LIN {X 0,Y 580.3,Z 452.202,A -85,B 0,C 180,E1 -1946.144,E2 -1946.144} C_VEL
LIN {X 0,Y 580.268,Z 452.203,A -85,B 0,C 180,E1 -1948.614,E2 -1948.614} C_VEL
LIN {X 0,Y 580.272,Z 452.198,A -85,B 0,C 180,E1 -1951.022,E2 -1951.022} C_VEL
LIN {X 0,Y 580.272,Z 452.198,A -85,B 0,C 180,E1 -1953.666,E2 -1953.666} C_VEL
LIN {X 0,Y 580.251,Z 452.21,A -85,B 0,C 180,E1 -1956.441,E2 -1956.441} C_VEL
LIN {X 0,Y 580.254,Z 452.2,A -85,B 0,C 180,E1 -1959.436,E2 -1959.436} C_VEL
LIN {X 0,Y 580.242,Z 452.202,A -85,B 0,C 180,E1 -1961.644,E2 -1961.644} C_VEL
LIN {X 0,Y 580.251,Z 452.202,A -85,B 0,C 180,E1 -1963.825,E2 -1963.825} C_VEL
LIN {X 0,Y 580.255,Z 452.206,A -85,B 0,C 180,E1 -1966.695,E2 -1966.695} C_VEL
LIN {X 0,Y 580.293,Z 452.195,A -85,B 0,C 180,E1 -1969.533,E2 -1969.533} C_VEL
LIN {X 0,Y 580.321,Z 452.199,A -85,B 0,C 180,E1 -1972.344,E2 -1972.344} C_VEL
LIN {X 0,Y 580.315,Z 452.194,A -85,B 0,C 180,E1 -1975.137,E2 -1975.137} C_VEL
LIN {X 0,Y 580.312,Z 452.194,A -85,B 0,C 180,E1 -1977.918,E2 -1977.918} C_VEL
LIN {X 0,Y 580.36,Z 452.195,A -85,B 0,C 180,E1 -1980.694,E2 -1980.694} C_VEL
LIN {X 0,Y 580.267,Z 452.198,A -85,B 0,C 180,E1 -1983.472,E2 -1983.472} C_VEL
LIN {X 0,Y 580.306,Z 452.193,A -85,B 0,C 180,E1 -1985.56,E2 -1985.56} C_VEL
LIN {X 0,Y 580.319,Z 452.198,A -85,B 0,C 180,E1 -1988.356,E2 -1988.356} C_VEL
LIN {X 0,Y 580.319,Z 452.193,A -85,B 0,C 180,E1 -1991.208,E2 -1991.208} C_VEL
LIN {X 0,Y 580.3,Z 452.199,A -85,B 0,C 180,E1 -1994.339,E2 -1994.339} C_VEL
LIN {X 0,Y 580.298,Z 452.201,A -85,B 0,C 180,E1 -1996.914,E2 -1996.914} C_VEL
LIN {X 0,Y 580.293,Z 452.195,A -85,B 0,C 180,E1 -1999.822,E2 -1999.822} C_VEL
LIN {X 0,Y 580.272,Z 452.199,A -85,B 0,C 180,E1 -2001.35,E2 -2001.35} C_VEL
LIN {X 0,Y 579.575,Z 452.286,A -85,B 0,C 180,E1 -2001.929,E2 -2001.929} C_VEL
LIN {X 0,Y 576.696,Z 452.651,A -85,B 0,C 180,E1 -2002.869,E2 -2002.869} C_VEL
LIN {X 0,Y 574.301,Z 452.945,A -85,B 0,C 180,E1 -2003.625,E2 -2003.625} C_VEL
LIN {X 0,Y 573.303,Z 453.068,A -85,B 0,C 180,E1 -2004.209,E2 -2004.209} C_VEL
LIN {X 0,Y 573.237,Z 453.079,A -85,B 0,C 180,E1 -2004.406,E2 -2004.406} C_VEL
LIN {X 0,Y 573.242,Z 453.08,A -85,B 0,C 180,E1 -2006.976,E2 -2006.976} C_VEL
LIN {X 0,Y 573.236,Z 453.075,A -85,B 0,C 180,E1 -2009.489,E2 -2009.489} C_VEL
LIN {X 0,Y 573.243,Z 453.075,A -85,B 0,C 180,E1 -2012.23,E2 -2012.23} C_VEL
LIN {X 0,Y 573.241,Z 453.084,A -85,B 0,C 180,E1 -2014.775,E2 -2014.775} C_VEL
LIN {X 0,Y 573.241,Z 453.078,A -85,B 0,C 180,E1 -2017.167,E2 -2017.167} C_VEL
LIN {X 0,Y 573.236,Z 453.074,A -85,B 0,C 180,E1 -2019.608,E2 -2019.608} C_VEL
LIN {X 0,Y 573.232,Z 453.081,A -85,B 0,C 180,E1 -2022.643,E2 -2022.643} C_VEL
LIN {X 0,Y 573.228,Z 453.075,A -85,B 0,C 180,E1 -2025.668,E2 -2025.668} C_VEL
LIN {X 0,Y 573.251,Z 453.077,A -85,B 0,C 180,E1 -2028.547,E2 -2028.547} C_VEL
LIN {X 0,Y 573.241,Z 453.078,A -85,B 0,C 180,E1 -2031.3,E2 -2031.3} C_VEL
LIN {X 0,Y 573.234,Z 453.074,A -85,B 0,C 180,E1 -2034.015,E2 -2034.015} C_VEL
LIN {X 0,Y 573.276,Z 453.072,A -85,B 0,C 180,E1 -2036.52,E2 -2036.52} C_VEL
LIN {X 0,Y 573.233,Z 453.083,A -85,B 0,C 180,E1 -2039.117,E2 -2039.117} C_VEL
LIN {X 0,Y 573.258,Z 453.071,A -85,B 0,C 180,E1 -2041.969,E2 -2041.969} C_VEL
LIN {X 0,Y 573.248,Z 453.076,A -85,B 0,C 180,E1 -2044.591,E2 -2044.591} C_VEL
LIN {X 0,Y 573.232,Z 453.076,A -85,B 0,C 180,E1 -2047.663,E2 -2047.663} C_VEL
LIN {X 0,Y 573.273,Z 453.074,A -85,B 0,C 180,E1 -2050.729,E2 -2050.729} C_VEL
LIN {X 0,Y 573.255,Z 453.074,A -85,B 0,C 180,E1 -2053.623,E2 -2053.623} C_VEL
LIN {X 0,Y 573.27,Z 453.071,A -85,B 0,C 180,E1 -2055.808,E2 -2055.808} C_VEL
LIN {X 0,Y 573.26,Z 453.075,A -85,B 0,C 180,E1 -2058.746,E2 -2058.746} C_VEL
LIN {X 0,Y 573.288,Z 453.073,A -85,B 0,C 180,E1 -2061.542,E2 -2061.542} C_VEL
LIN {X 0,Y 573.295,Z 453.068,A -85,B 0,C 180,E1 -2064.373,E2 -2064.373} C_VEL
LIN {X 0,Y 573.313,Z 453.068,A -85,B 0,C 180,E1 -2067.894,E2 -2067.894} C_VEL
LIN {X 0,Y 573.342,Z 453.273,A -85,B 0,C 180,E1 -2070.462,E2 -2070.462} C_VEL
LIN {X 0,Y 573.575,Z 454.38,A -85,B 0,C 180,E1 -2070.572,E2 -2070.572} C_VEL
LIN {X 0,Y 574.043,Z 456.439,A -85,B 0,C 180,E1 -2070.615,E2 -2070.615} C_VEL
LIN {X 0,Y 573.909,Z 533.892,A -85,B 0,C 180,E1 -2071.602,E2 -2071.602} C_VEL
LIN {X 0,Y 573.777,Z 547.056,A -85,B 0,C 180,E1 -2071.91,E2 -2071.91} C_VEL
LIN {X 0,Y 573.683,Z 559.086,A -85,B 0,C 180,E1 -2072.327,E2 -2072.327} C_VEL
LIN {X 0,Y 573.567,Z 571.273,A -85,B 0,C 180,E1 -2072.898,E2 -2072.898} C_VEL
LIN {X 0,Y 573.429,Z 582.799,A -85,B 0,C 180,E1 -2073.602,E2 -2073.602} C_VEL
LIN {X 0,Y 573.315,Z 593.186,A -85,B 0,C 180,E1 -2074.395,E2 -2074.395} C_VEL
LIN {X 0,Y 573.24,Z 602.582,A -85,B 0,C 180,E1 -2075.277,E2 -2075.277} C_VEL
LIN {X 0,Y 573.148,Z 611.669,A -85,B 0,C 180,E1 -2076.337,E2 -2076.337} C_VEL
LIN {X 0,Y 573.107,Z 619.017,A -85,B 0,C 180,E1 -2077.399,E2 -2077.399} C_VEL
LIN {X 0,Y 573.056,Z 624.934,A -85,B 0,C 180,E1 -2078.464,E2 -2078.464} C_VEL
LIN {X 0,Y 572.993,Z 629.615,A -85,B 0,C 180,E1 -2079.532,E2 -2079.532} C_VEL
LIN {X 0,Y 573.009,Z 633.181,A -85,B 0,C 180,E1 -2080.603,E2 -2080.603} C_VEL
LIN {X 0,Y 572.975,Z 634.995,A -85,B 0,C 180,E1 -2081.319,E2 -2081.319} C_VEL
LIN {X 0,Y 572.946,Z 636.36,A -85,B 0,C 180,E1 -2082.037,E2 -2082.037} C_VEL
LIN {X 0,Y 572.945,Z 637.318,A -85,B 0,C 180,E1 -2082.757,E2 -2082.757} C_VEL
LIN {X 0,Y 572.968,Z 637.871,A -85,B 0,C 180,E1 -2083.478,E2 -2083.478} C_VEL
LIN {X 0,Y 572.942,Z 637.951,A -85,B 0,C 180,E1 -2084.292,E2 -2084.292} C_VEL
LIN {X 0,Y 572.916,Z 636.947,A -85,B 0,C 180,E1 -2085.658,E2 -2085.658} C_VEL
LIN {X 0,Y 572.943,Z 634.69,A -85,B 0,C 180,E1 -2086.906,E2 -2086.906} C_VEL
LIN {X 0,Y 572.997,Z 630.813,A -85,B 0,C 180,E1 -2088.227,E2 -2088.227} C_VEL
LIN {X 0,Y 573.042,Z 626.292,A -85,B 0,C 180,E1 -2089.339,E2 -2089.339} C_VEL
LIN {X 0,Y 573.065,Z 620.428,A -85,B 0,C 180,E1 -2090.459,E2 -2090.459} C_VEL
LIN {X 0,Y 573.128,Z 612.949,A -85,B 0,C 180,E1 -2091.586,E2 -2091.586} C_VEL
LIN {X 0,Y 573.206,Z 605.19,A -85,B 0,C 180,E1 -2092.53,E2 -2092.53} C_VEL
LIN {X 0,Y 573.307,Z 596.066,A -85,B 0,C 180,E1 -2093.441,E2 -2093.441} C_VEL
LIN {X 0,Y 573.369,Z 586.243,A -85,B 0,C 180,E1 -2094.245,E2 -2094.245} C_VEL
LIN {X 0,Y 573.53,Z 575.819,A -85,B 0,C 180,E1 -2094.935,E2 -2094.935} C_VEL
LIN {X 0,Y 573.646,Z 564.277,A -85,B 0,C 180,E1 -2095.538,E2 -2095.538} C_VEL
LIN {X 0,Y 573.712,Z 552.108,A -85,B 0,C 180,E1 -2096.022,E2 -2096.022} C_VEL
LIN {X 0,Y 573.878,Z 538.874,A -85,B 0,C 180,E1 -2096.39,E2 -2096.39} C_VEL
LIN {X 0,Y 573.912,Z 524.024,A -85,B 0,C 180,E1 -2096.628,E2 -2096.628} C_VEL
LIN {X 0,Y 573.945,Z 455.681,A -85,B 0,C 180,E1 -2097.487,E2 -2097.487} C_VEL
LIN {X 0,Y 573.406,Z 453.736,A -85,B 0,C 180,E1 -2097.562,E2 -2097.562} C_VEL
LIN {X 0,Y 573.286,Z 453.1,A -85,B 0,C 180,E1 -2097.717,E2 -2097.717} C_VEL
LIN {X 0,Y 573.249,Z 453.077,A -85,B 0,C 180,E1 -2100.177,E2 -2100.177} C_VEL
LIN {X 0,Y 573.257,Z 453.079,A -85,B 0,C 180,E1 -2102.646,E2 -2102.646} C_VEL
LIN {X 0,Y 573.21,Z 453.083,A -85,B 0,C 180,E1 -2105.189,E2 -2105.189} C_VEL
LIN {X 0,Y 573.237,Z 453.075,A -85,B 0,C 180,E1 -2107.809,E2 -2107.809} C_VEL
LIN {X 0,Y 573.248,Z 453.077,A -85,B 0,C 180,E1 -2110.526,E2 -2110.526} C_VEL
LIN {X 0,Y 573.241,Z 453.077,A -85,B 0,C 180,E1 -2113.36,E2 -2113.36} C_VEL
LIN {X 0,Y 573.24,Z 453.081,A -85,B 0,C 180,E1 -2116.641,E2 -2116.641} C_VEL
LIN {X 0,Y 573.249,Z 453.076,A -85,B 0,C 180,E1 -2119.476,E2 -2119.476} C_VEL
LIN {X 0,Y 573.236,Z 453.078,A -85,B 0,C 180,E1 -2122.193,E2 -2122.193} C_VEL
LIN {X 0,Y 573.303,Z 453.256,A -85,B 0,C 180,E1 -2124.007,E2 -2124.007} C_VEL
LIN {X 0,Y 573.988,Z 458.626,A -85,B 0,C 180,E1 -2124.867,E2 -2124.867} C_VEL
LIN {X 0,Y 573.753,Z 477.734,A -85,B 0,C 180,E1 -2127.694,E2 -2127.694} C_VEL
LIN {X 0,Y 573.532,Z 498.047,A -85,B 0,C 180,E1 -2130.649,E2 -2130.649} C_VEL
LIN {X 0,Y 573.409,Z 515.835,A -85,B 0,C 180,E1 -2133.178,E2 -2133.178} C_VEL
LIN {X 0,Y 573.919,Z 519.481,A -85,B 0,C 180,E1 -2133.272,E2 -2133.272} C_VEL
LIN {X 0,Y 573.884,Z 623.362,A -85,B 0,C 180,E1 -2134.596,E2 -2134.596} C_VEL
LIN {X 0,Y 573.834,Z 636.448,A -85,B 0,C 180,E1 -2134.891,E2 -2134.891} C_VEL
LIN {X 0,Y 573.662,Z 649.183,A -85,B 0,C 180,E1 -2135.331,E2 -2135.331} C_VEL
LIN {X 0,Y 573.566,Z 660.509,A -85,B 0,C 180,E1 -2135.861,E2 -2135.861} C_VEL
LIN {X 0,Y 573.471,Z 671.716,A -85,B 0,C 180,E1 -2136.527,E2 -2136.527} C_VEL
LIN {X 0,Y 573.363,Z 681.861,A -85,B 0,C 180,E1 -2137.288,E2 -2137.288} C_VEL
LIN {X 0,Y 573.26,Z 690.215,A -85,B 0,C 180,E1 -2138.043,E2 -2138.043} C_VEL
LIN {X 0,Y 573.163,Z 698.524,A -85,B 0,C 180,E1 -2138.944,E2 -2138.944} C_VEL
LIN {X 0,Y 573.101,Z 707.128,A -85,B 0,C 180,E1 -2140.105,E2 -2140.105} C_VEL
LIN {X 0,Y 573.074,Z 713.021,A -85,B 0,C 180,E1 -2141.097,E2 -2141.097} C_VEL
LIN {X 0,Y 572.995,Z 718.04,A -85,B 0,C 180,E1 -2142.144,E2 -2142.144} C_VEL
LIN {X 0,Y 572.999,Z 721.552,A -85,B 0,C 180,E1 -2143.079,E2 -2143.079} C_VEL
LIN {X 0,Y 572.936,Z 725.046,A -85,B 0,C 180,E1 -2144.344,E2 -2144.344} C_VEL
LIN {X 0,Y 572.91,Z 726.425,A -85,B 0,C 180,E1 -2145.072,E2 -2145.072} C_VEL
LIN {X 0,Y 572.983,Z 727.347,A -85,B 0,C 180,E1 -2145.8,E2 -2145.8} C_VEL
LIN {X 0,Y 572.971,Z 727.86,A -85,B 0,C 180,E1 -2146.523,E2 -2146.523} C_VEL
LIN {X 0,Y 572.946,Z 727.962,A -85,B 0,C 180,E1 -2147.245,E2 -2147.245} C_VEL
LIN {X 0,Y 572.949,Z 727.648,A -85,B 0,C 180,E1 -2147.964,E2 -2147.964} C_VEL
LIN {X 0,Y 572.989,Z 726.625,A -85,B 0,C 180,E1 -2148.888,E2 -2148.888} C_VEL
LIN {X 0,Y 572.979,Z 724.172,A -85,B 0,C 180,E1 -2150.112,E2 -2150.112} C_VEL
LIN {X 0,Y 573.003,Z 720.956,A -85,B 0,C 180,E1 -2151.181,E2 -2151.181} C_VEL
LIN {X 0,Y 573.025,Z 716.709,A -85,B 0,C 180,E1 -2152.247,E2 -2152.247} C_VEL
LIN {X 0,Y 573.097,Z 710.892,A -85,B 0,C 180,E1 -2153.379,E2 -2153.379} C_VEL
LIN {X 0,Y 573.084,Z 703.217,A -85,B 0,C 180,E1 -2154.547,E2 -2154.547} C_VEL
LIN {X 0,Y 573.216,Z 694.51,A -85,B 0,C 180,E1 -2155.605,E2 -2155.605} C_VEL
LIN {X 0,Y 573.325,Z 684.562,A -85,B 0,C 180,E1 -2156.574,E2 -2156.574} C_VEL
LIN {X 0,Y 573.451,Z 674.523,A -85,B 0,C 180,E1 -2157.366,E2 -2157.366} C_VEL
LIN {X 0,Y 573.54,Z 663.481,A -85,B 0,C 180,E1 -2158.069,E2 -2158.069} C_VEL
LIN {X 0,Y 573.619,Z 651.996,A -85,B 0,C 180,E1 -2158.64,E2 -2158.64} C_VEL
LIN {X 0,Y 573.797,Z 640.3,A -85,B 0,C 180,E1 -2159.079,E2 -2159.079} C_VEL
LIN {X 0,Y 573.877,Z 628.037,A -85,B 0,C 180,E1 -2159.408,E2 -2159.408} C_VEL
LIN {X 0,Y 573.934,Z 610.521,A -85,B 0,C 180,E1 -2159.671,E2 -2159.671} C_VEL
LIN {X 0,Y 573.963,Z 519.91,A -85,B 0,C 180,E1 -2160.811,E2 -2160.811} C_VEL
LIN {X 0,Y 573.365,Z 516.022,A -85,B 0,C 180,E1 -2160.9,E2 -2160.9} C_VEL
LIN {X 0,Y 573.525,Z 500.068,A -85,B 0,C 180,E1 -2163.161,E2 -2163.161} C_VEL
LIN {X 0,Y 573.751,Z 479.559,A -85,B 0,C 180,E1 -2166.153,E2 -2166.153} C_VEL
LIN {X 0,Y 573.949,Z 460.49,A -85,B 0,C 180,E1 -2168.982,E2 -2168.982} C_VEL
LIN {X 0,Y 573.787,Z 455.793,A -85,B 0,C 180,E1 -2169.696,E2 -2169.696} C_VEL
LIN {X 0,Y 573.253,Z 453.181,A -85,B 0,C 180,E1 -2170.151,E2 -2170.151} C_VEL
LIN {X 0,Y 573.218,Z 453.082,A -85,B 0,C 180,E1 -2172.75,E2 -2172.75} C_VEL
LIN {X 0,Y 573.222,Z 453.084,A -85,B 0,C 180,E1 -2174.92,E2 -2174.92} C_VEL
LIN {X 0,Y 573.222,Z 453.078,A -85,B 0,C 180,E1 -2177.849,E2 -2177.849} C_VEL
LIN {X 0,Y 573.237,Z 453.075,A -85,B 0,C 180,E1 -2180.077,E2 -2180.077} C_VEL
LIN {X 0,Y 573.227,Z 453.078,A -85,B 0,C 180,E1 -2182.338,E2 -2182.338} C_VEL
LIN {X 0,Y 573.247,Z 453.077,A -85,B 0,C 180,E1 -2185.411,E2 -2185.411} C_VEL
LIN {X 0,Y 573.252,Z 453.074,A -85,B 0,C 180,E1 -2188.027,E2 -2188.027} C_VEL
LIN {X 0,Y 573.246,Z 453.075,A -85,B 0,C 180,E1 -2190.176,E2 -2190.176} C_VEL
LIN {X 0,Y 573.262,Z 453.08,A -85,B 0,C 180,E1 -2192.645,E2 -2192.645} C_VEL
LIN {X 0,Y 573.217,Z 453.08,A -85,B 0,C 180,E1 -2195.187,E2 -2195.187} C_VEL
LIN {X 0,Y 573.242,Z 453.075,A -85,B 0,C 180,E1 -2197.807,E2 -2197.807} C_VEL
LIN {X 0,Y 573.253,Z 453.082,A -85,B 0,C 180,E1 -2200.525,E2 -2200.525} C_VEL
LIN {X 0,Y 573.244,Z 453.074,A -85,B 0,C 180,E1 -2203.359,E2 -2203.359} C_VEL
LIN {X 0,Y 573.244,Z 453.08,A -85,B 0,C 180,E1 -2206.64,E2 -2206.64} C_VEL
LIN {X 0,Y 573.252,Z 453.074,A -85,B 0,C 180,E1 -2209.474,E2 -2209.474} C_VEL
LIN {X 0,Y 573.237,Z 453.079,A -85,B 0,C 180,E1 -2212.191,E2 -2212.191} C_VEL
LIN {X 0,Y 573.23,Z 453.075,A -85,B 0,C 180,E1 -2215.23,E2 -2215.23} C_VEL
LIN {X 0,Y 573.244,Z 453.083,A -85,B 0,C 180,E1 -2218.184,E2 -2218.184} C_VEL
LIN {X 0,Y 573.249,Z 453.078,A -85,B 0,C 180,E1 -2220.632,E2 -2220.632} C_VEL
LIN {X 0,Y 573.25,Z 453.246,A -85,B 0,C 180,E1 -2222.789,E2 -2222.789} C_VEL
LIN {X 0,Y 574.825,Z 459.837,A -85,B 0,C 180,E1 -2223.596,E2 -2223.596} C_VEL
LIN {X 0,Y 574.676,Z 474.923,A -85,B 0,C 180,E1 -2225.279,E2 -2225.279} C_VEL
LIN {X 0,Y 574.383,Z 498.182,A -85,B 0,C 180,E1 -2227.898,E2 -2227.898} C_VEL
LIN {X 0,Y 574.009,Z 523.496,A -85,B 0,C 180,E1 -2230.695,E2 -2230.695} C_VEL
LIN {X 0,Y 573.744,Z 550.5,A -85,B 0,C 180,E1 -2233.635,E2 -2233.635} C_VEL
LIN {X 0,Y 573.549,Z 573.847,A -85,B 0,C 180,E1 -2236.13,E2 -2236.13} C_VEL
LIN {X 0,Y 574.086,Z 579.633,A -85,B 0,C 180,E1 -2236.233,E2 -2236.233} C_VEL
LIN {X 0,Y 573.88,Z 683.89,A -85,B 0,C 180,E1 -2237.556,E2 -2237.556} C_VEL
LIN {X 0,Y 573.805,Z 697.182,A -85,B 0,C 180,E1 -2237.869,E2 -2237.869} C_VEL
LIN {X 0,Y 573.707,Z 710.123,A -85,B 0,C 180,E1 -2238.324,E2 -2238.324} C_VEL
LIN {X 0,Y 573.581,Z 721.716,A -85,B 0,C 180,E1 -2238.878,E2 -2238.878} C_VEL
LIN {X 0,Y 573.438,Z 733.187,A -85,B 0,C 180,E1 -2239.584,E2 -2239.584} C_VEL
LIN {X 0,Y 573.331,Z 743.586,A -85,B 0,C 180,E1 -2240.384,E2 -2240.384} C_VEL
LIN {X 0,Y 573.24,Z 752.101,A -85,B 0,C 180,E1 -2241.183,E2 -2241.183} C_VEL
LIN {X 0,Y 573.162,Z 759.951,A -85,B 0,C 180,E1 -2242.07,E2 -2242.07} C_VEL
LIN {X 0,Y 573.074,Z 767.948,A -85,B 0,C 180,E1 -2243.185,E2 -2243.185} C_VEL
LIN {X 0,Y 573.07,Z 774.674,A -85,B 0,C 180,E1 -2244.369,E2 -2244.369} C_VEL
LIN {X 0,Y 573.029,Z 779.367,A -85,B 0,C 180,E1 -2245.426,E2 -2245.426} C_VEL
LIN {X 0,Y 573.022,Z 782.954,A -85,B 0,C 180,E1 -2246.483,E2 -2246.483} C_VEL
LIN {X 0,Y 572.959,Z 784.806,A -85,B 0,C 180,E1 -2247.187,E2 -2247.187} C_VEL
LIN {X 0,Y 572.939,Z 786.197,A -85,B 0,C 180,E1 -2247.89,E2 -2247.89} C_VEL
LIN {X 0,Y 572.94,Z 787.784,A -85,B 0,C 180,E1 -2249.296,E2 -2249.296} C_VEL
LIN {X 0,Y 572.938,Z 788,A -85,B 0,C 180,E1 -2249.999,E2 -2249.999} C_VEL
LIN {X 0,Y 572.946,Z 787.187,A -85,B 0,C 180,E1 -2251.405,E2 -2251.405} C_VEL
LIN {X 0,Y 572.939,Z 786.202,A -85,B 0,C 180,E1 -2252.108,E2 -2252.108} C_VEL
LIN {X 0,Y 572.959,Z 784.813,A -85,B 0,C 180,E1 -2252.811,E2 -2252.811} C_VEL
LIN {X 0,Y 573.014,Z 781.9,A -85,B 0,C 180,E1 -2253.867,E2 -2253.867} C_VEL
LIN {X 0,Y 572.962,Z 777.954,A -85,B 0,C 180,E1 -2254.924,E2 -2254.924} C_VEL
LIN {X 0,Y 573.064,Z 771.884,A -85,B 0,C 180,E1 -2256.159,E2 -2256.159} C_VEL
LIN {X 0,Y 573.119,Z 765.246,A -85,B 0,C 180,E1 -2257.22,E2 -2257.22} C_VEL
LIN {X 0,Y 573.2,Z 757.001,A -85,B 0,C 180,E1 -2258.282,E2 -2258.282} C_VEL
LIN {X 0,Y 573.286,Z 748.552,A -85,B 0,C 180,E1 -2259.169,E2 -2259.169} C_VEL
LIN {X 0,Y 573.413,Z 738.114,A -85,B 0,C 180,E1 -2260.057,E2 -2260.057} C_VEL
LIN {X 0,Y 573.533,Z 727.792,A -85,B 0,C 180,E1 -2260.768,E2 -2260.768} C_VEL
LIN {X 0,Y 573.626,Z 716.614,A -85,B 0,C 180,E1 -2261.384,E2 -2261.384} C_VEL
LIN {X 0,Y 573.712,Z 704.805,A -85,B 0,C 180,E1 -2261.884,E2 -2261.884} C_VEL
LIN {X 0,Y 573.808,Z 691.402,A -85,B 0,C 180,E1 -2262.286,E2 -2262.286} C_VEL
LIN {X 0,Y 573.939,Z 678.178,A -85,B 0,C 180,E1 -2262.53,E2 -2262.53} C_VEL
LIN {X 0,Y 573.952,Z 577.143,A -85,B 0,C 180,E1 -2263.802,E2 -2263.802} C_VEL
LIN {X 0,Y 573.549,Z 573.912,A -85,B 0,C 180,E1 -2263.868,E2 -2263.868} C_VEL
LIN {X 0,Y 573.786,Z 547.279,A -85,B 0,C 180,E1 -2266.727,E2 -2266.727} C_VEL
LIN {X 0,Y 574.046,Z 522.052,A -85,B 0,C 180,E1 -2269.488,E2 -2269.488} C_VEL
LIN {X 0,Y 574.391,Z 496.849,A -85,B 0,C 180,E1 -2272.289,E2 -2272.289} C_VEL
LIN {X 0,Y 574.785,Z 472.305,A -85,B 0,C 180,E1 -2275.065,E2 -2275.065} C_VEL
LIN {X 0,Y 574.881,Z 460.282,A -85,B 0,C 180,E1 -2276.408,E2 -2276.408} C_VEL
LIN {X 0,Y 573.226,Z 453.177,A -85,B 0,C 180,E1 -2277.296,E2 -2277.296} C_VEL
LIN {X 0,Y 573.225,Z 453.086,A -85,B 0,C 180,E1 -2280.176,E2 -2280.176} C_VEL
LIN {X 0,Y 573.246,Z 453.077,A -85,B 0,C 180,E1 -2282.644,E2 -2282.644} C_VEL
LIN {X 0,Y 573.181,Z 453.082,A -85,B 0,C 180,E1 -2285.188,E2 -2285.188} C_VEL
LIN {X 0,Y 573.212,Z 453.081,A -85,B 0,C 180,E1 -2287.807,E2 -2287.807} C_VEL
LIN {X 0,Y 573.237,Z 453.079,A -85,B 0,C 180,E1 -2290.524,E2 -2290.524} C_VEL
LIN {X 0,Y 573.199,Z 453.079,A -85,B 0,C 180,E1 -2293.361,E2 -2293.361} C_VEL
LIN {X 0,Y 573.225,Z 453.084,A -85,B 0,C 180,E1 -2296.331,E2 -2296.331} C_VEL
LIN {X 0,Y 573.235,Z 453.075,A -85,B 0,C 180,E1 -2299.474,E2 -2299.474} C_VEL
LIN {X 0,Y 573.218,Z 453.086,A -85,B 0,C 180,E1 -2302.191,E2 -2302.191} C_VEL
LIN {X 0,Y 573.22,Z 453.076,A -85,B 0,C 180,E1 -2305.228,E2 -2305.228} C_VEL
LIN {X 0,Y 573.238,Z 453.076,A -85,B 0,C 180,E1 -2307.771,E2 -2307.771} C_VEL
LIN {X 0,Y 573.243,Z 453.078,A -85,B 0,C 180,E1 -2310.633,E2 -2310.633} C_VEL
LIN {X 0,Y 573.207,Z 453.079,A -85,B 0,C 180,E1 -2313.022,E2 -2313.022} C_VEL
LIN {X 0,Y 573.223,Z 453.076,A -85,B 0,C 180,E1 -2315.363,E2 -2315.363} C_VEL
LIN {X 0,Y 573.211,Z 453.078,A -85,B 0,C 180,E1 -2317.661,E2 -2317.661} C_VEL
LIN {X 0,Y 573.254,Z 453.078,A -85,B 0,C 180,E1 -2320.669,E2 -2320.669} C_VEL
LIN {X 0,Y 573.226,Z 453.076,A -85,B 0,C 180,E1 -2323.621,E2 -2323.621} C_VEL
LIN {X 0,Y 573.212,Z 453.086,A -85,B 0,C 180,E1 -2326.529,E2 -2326.529} C_VEL
LIN {X 0,Y 573.271,Z 453.076,A -85,B 0,C 180,E1 -2328.733,E2 -2328.733} C_VEL
LIN {X 0,Y 573.239,Z 453.074,A -85,B 0,C 180,E1 -2331.54,E2 -2331.54} C_VEL
LIN {X 0,Y 573.276,Z 453.077,A -85,B 0,C 180,E1 -2334.371,E2 -2334.371} C_VEL
LIN {X 0,Y 573.29,Z 453.068,A -85,B 0,C 180,E1 -2337.189,E2 -2337.189} C_VEL
LIN {X 0,Y 573.297,Z 453.069,A -85,B 0,C 180,E1 -2340,E2 -2340} C_VEL
LIN {X 0,Y 573.303,Z 453.072,A -85,B 0,C 180,E1 -2342.81,E2 -2342.81} C_VEL
LIN {X 0,Y 573.273,Z 453.069,A -85,B 0,C 180,E1 -2345.628,E2 -2345.628} C_VEL
LIN {X 0,Y 573.292,Z 453.075,A -85,B 0,C 180,E1 -2348.459,E2 -2348.459} C_VEL
LIN {X 0,Y 573.285,Z 453.069,A -85,B 0,C 180,E1 -2351.311,E2 -2351.311} C_VEL
LIN {X 0,Y 573.267,Z 453.077,A -85,B 0,C 180,E1 -2354.425,E2 -2354.425} C_VEL
LIN {X 0,Y 573.244,Z 453.076,A -85,B 0,C 180,E1 -2357.112,E2 -2357.112} C_VEL
LIN {X 0,Y 573.243,Z 453.075,A -85,B 0,C 180,E1 -2360.077,E2 -2360.077} C_VEL
LIN {X 0,Y 573.224,Z 453.08,A -85,B 0,C 180,E1 -2362.338,E2 -2362.338} C_VEL
LIN {X 0,Y 573.237,Z 453.079,A -85,B 0,C 180,E1 -2364.406,E2 -2364.406} C_VEL
LIN {X 0,Y 572.612,Z 453.163,A -85,B 0,C 180,E1 -2364.993,E2 -2364.993} C_VEL
LIN {X 0,Y 569.77,Z 453.517,A -85,B 0,C 180,E1 -2365.944,E2 -2365.944} C_VEL
LIN {X 0,Y 567.34,Z 453.819,A -85,B 0,C 180,E1 -2366.71,E2 -2366.71} C_VEL
LIN {X 0,Y 566.288,Z 453.942,A -85,B 0,C 180,E1 -2367.301,E2 -2367.301} C_VEL
LIN {X 0,Y 566.2,Z 453.951,A -85,B 0,C 180,E1 -2367.501,E2 -2367.501} C_VEL
LIN {X 0,Y 566.176,Z 453.961,A -85,B 0,C 180,E1 -2370.593,E2 -2370.593} C_VEL
LIN {X 0,Y 566.216,Z 453.954,A -85,B 0,C 180,E1 -2373.102,E2 -2373.102} C_VEL
LIN {X 0,Y 566.198,Z 453.951,A -85,B 0,C 180,E1 -2375.689,E2 -2375.689} C_VEL
LIN {X 0,Y 566.204,Z 453.956,A -85,B 0,C 180,E1 -2378.56,E2 -2378.56} C_VEL
LIN {X 0,Y 566.201,Z 453.956,A -85,B 0,C 180,E1 -2381.137,E2 -2381.137} C_VEL
LIN {X 0,Y 566.189,Z 453.952,A -85,B 0,C 180,E1 -2384.036,E2 -2384.036} C_VEL
LIN {X 0,Y 566.2,Z 453.958,A -85,B 0,C 180,E1 -2387.083,E2 -2387.083} C_VEL
LIN {X 0,Y 566.217,Z 453.948,A -85,B 0,C 180,E1 -2389.804,E2 -2389.804} C_VEL
LIN {X 0,Y 566.19,Z 453.956,A -85,B 0,C 180,E1 -2392.6,E2 -2392.6} C_VEL
LIN {X 0,Y 566.205,Z 453.956,A -85,B 0,C 180,E1 -2395.184,E2 -2395.184} C_VEL
LIN {X 0,Y 566.229,Z 453.947,A -85,B 0,C 180,E1 -2397.745,E2 -2397.745} C_VEL
LIN {X 0,Y 566.196,Z 453.952,A -85,B 0,C 180,E1 -2400.329,E2 -2400.329} C_VEL
LIN {X 0,Y 566.213,Z 453.953,A -85,B 0,C 180,E1 -2402.663,E2 -2402.663} C_VEL
LIN {X 0,Y 566.23,Z 453.957,A -85,B 0,C 180,E1 -2405.04,E2 -2405.04} C_VEL
LIN {X 0,Y 566.189,Z 453.952,A -85,B 0,C 180,E1 -2408.139,E2 -2408.139} C_VEL
LIN {X 0,Y 566.231,Z 453.95,A -85,B 0,C 180,E1 -2410.613,E2 -2410.613} C_VEL
LIN {X 0,Y 566.216,Z 453.953,A -85,B 0,C 180,E1 -2413.414,E2 -2413.414} C_VEL
LIN {X 0,Y 566.196,Z 453.952,A -85,B 0,C 180,E1 -2416.36,E2 -2416.36} C_VEL
LIN {X 0,Y 566.231,Z 453.95,A -85,B 0,C 180,E1 -2418.676,E2 -2418.676} C_VEL
LIN {X 0,Y 566.231,Z 453.953,A -85,B 0,C 180,E1 -2421.436,E2 -2421.436} C_VEL
LIN {X 0,Y 566.264,Z 453.944,A -85,B 0,C 180,E1 -2424.303,E2 -2424.303} C_VEL
LIN {X 0,Y 566.283,Z 453.944,A -85,B 0,C 180,E1 -2427.867,E2 -2427.867} C_VEL
LIN {X 0,Y 566.31,Z 454.125,A -85,B 0,C 180,E1 -2430.29,E2 -2430.29} C_VEL
LIN {X 0,Y 566.528,Z 455.107,A -85,B 0,C 180,E1 -2430.401,E2 -2430.401} C_VEL
LIN {X 0,Y 567.152,Z 458.178,A -85,B 0,C 180,E1 -2430.467,E2 -2430.467} C_VEL
LIN {X 0,Y 566.984,Z 534.945,A -85,B 0,C 180,E1 -2431.466,E2 -2431.466} C_VEL
LIN {X 0,Y 566.823,Z 548.471,A -85,B 0,C 180,E1 -2431.8,E2 -2431.8} C_VEL
LIN {X 0,Y 566.713,Z 561.146,A -85,B 0,C 180,E1 -2432.267,E2 -2432.267} C_VEL
LIN {X 0,Y 566.563,Z 572.786,A -85,B 0,C 180,E1 -2432.845,E2 -2432.845} C_VEL
LIN {X 0,Y 566.431,Z 584.027,A -85,B 0,C 180,E1 -2433.558,E2 -2433.558} C_VEL
LIN {X 0,Y 566.268,Z 594.208,A -85,B 0,C 180,E1 -2434.361,E2 -2434.361} C_VEL
LIN {X 0,Y 566.182,Z 604.185,A -85,B 0,C 180,E1 -2435.343,E2 -2435.343} C_VEL
LIN {X 0,Y 566.072,Z 613.002,A -85,B 0,C 180,E1 -2436.417,E2 -2436.417} C_VEL
LIN {X 0,Y 566.006,Z 620.1,A -85,B 0,C 180,E1 -2437.492,E2 -2437.492} C_VEL
LIN {X 0,Y 565.95,Z 625.779,A -85,B 0,C 180,E1 -2438.571,E2 -2438.571} C_VEL
LIN {X 0,Y 565.916,Z 630.262,A -85,B 0,C 180,E1 -2439.653,E2 -2439.653} C_VEL
LIN {X 0,Y 565.91,Z 633.663,A -85,B 0,C 180,E1 -2440.737,E2 -2440.737} C_VEL
LIN {X 0,Y 565.872,Z 635.358,A -85,B 0,C 180,E1 -2441.463,E2 -2441.463} C_VEL
LIN {X 0,Y 565.865,Z 636.64,A -85,B 0,C 180,E1 -2442.19,E2 -2442.19} C_VEL
LIN {X 0,Y 565.843,Z 637.505,A -85,B 0,C 180,E1 -2442.92,E2 -2442.92} C_VEL
LIN {X 0,Y 565.863,Z 637.919,A -85,B 0,C 180,E1 -2443.65,E2 -2443.65} C_VEL
LIN {X 0,Y 565.839,Z 637.93,A -85,B 0,C 180,E1 -2444.385,E2 -2444.385} C_VEL
LIN {X 0,Y 565.805,Z 637.539,A -85,B 0,C 180,E1 -2445.121,E2 -2445.121} C_VEL
LIN {X 0,Y 565.813,Z 636.698,A -85,B 0,C 180,E1 -2445.86,E2 -2445.86} C_VEL
LIN {X 0,Y 565.858,Z 634.564,A -85,B 0,C 180,E1 -2446.993,E2 -2446.993} C_VEL
LIN {X 0,Y 565.912,Z 631.476,A -85,B 0,C 180,E1 -2448.089,E2 -2448.089} C_VEL
LIN {X 0,Y 565.954,Z 626.736,A -85,B 0,C 180,E1 -2449.307,E2 -2449.307} C_VEL
LIN {X 0,Y 565.992,Z 620.447,A -85,B 0,C 180,E1 -2450.536,E2 -2450.536} C_VEL
LIN {X 0,Y 566.067,Z 613.847,A -85,B 0,C 180,E1 -2451.558,E2 -2451.558} C_VEL
LIN {X 0,Y 566.155,Z 605.216,A -85,B 0,C 180,E1 -2452.634,E2 -2452.634} C_VEL
LIN {X 0,Y 566.292,Z 595.681,A -85,B 0,C 180,E1 -2453.594,E2 -2453.594} C_VEL
LIN {X 0,Y 566.407,Z 584.993,A -85,B 0,C 180,E1 -2454.465,E2 -2454.465} C_VEL
LIN {X 0,Y 566.588,Z 573.655,A -85,B 0,C 180,E1 -2455.195,E2 -2455.195} C_VEL
LIN {X 0,Y 566.715,Z 561.126,A -85,B 0,C 180,E1 -2455.824,E2 -2455.824} C_VEL
LIN {X 0,Y 566.845,Z 548.527,A -85,B 0,C 180,E1 -2456.287,E2 -2456.287} C_VEL
LIN {X 0,Y 566.957,Z 536.159,A -85,B 0,C 180,E1 -2456.599,E2 -2456.599} C_VEL
LIN {X 0,Y 567.017,Z 513.749,A -85,B 0,C 180,E1 -2456.916,E2 -2456.916} C_VEL
LIN {X 0,Y 566.996,Z 456.753,A -85,B 0,C 180,E1 -2457.645,E2 -2457.645} C_VEL
LIN {X 0,Y 566.396,Z 454.785,A -85,B 0,C 180,E1 -2457.712,E2 -2457.712} C_VEL
LIN {X 0,Y 566.259,Z 454.013,A -85,B 0,C 180,E1 -2457.839,E2 -2457.839} C_VEL
LIN {X 0,Y 566.184,Z 453.962,A -85,B 0,C 180,E1 -2460.594,E2 -2460.594} C_VEL
LIN {X 0,Y 566.208,Z 453.957,A -85,B 0,C 180,E1 -2463.104,E2 -2463.104} C_VEL
LIN {X 0,Y 566.166,Z 453.957,A -85,B 0,C 180,E1 -2465.693,E2 -2465.693} C_VEL
LIN {X 0,Y 566.212,Z 453.955,A -85,B 0,C 180,E1 -2468.559,E2 -2468.559} C_VEL
LIN {X 0,Y 566.176,Z 453.959,A -85,B 0,C 180,E1 -2471.141,E2 -2471.141} C_VEL
LIN {X 0,Y 566.196,Z 453.952,A -85,B 0,C 180,E1 -2474.037,E2 -2474.037} C_VEL
LIN {X 0,Y 566.205,Z 453.957,A -85,B 0,C 180,E1 -2477.084,E2 -2477.084} C_VEL
LIN {X 0,Y 566.217,Z 453.953,A -85,B 0,C 180,E1 -2480.315,E2 -2480.315} C_VEL
LIN {X 0,Y 566.219,Z 453.957,A -85,B 0,C 180,E1 -2483.432,E2 -2483.432} C_VEL
LIN {X 0,Y 566.24,Z 454.107,A -85,B 0,C 180,E1 -2483.848,E2 -2483.848} C_VEL
LIN {X 0,Y 567.047,Z 459.229,A -85,B 0,C 180,E1 -2484.673,E2 -2484.673} C_VEL
LIN {X 0,Y 566.814,Z 478.469,A -85,B 0,C 180,E1 -2487.557,E2 -2487.557} C_VEL
LIN {X 0,Y 566.537,Z 499.535,A -85,B 0,C 180,E1 -2490.659,E2 -2490.659} C_VEL
LIN {X 0,Y 566.396,Z 515.959,A -85,B 0,C 180,E1 -2493.012,E2 -2493.012} C_VEL
LIN {X 0,Y 567.15,Z 521.083,A -85,B 0,C 180,E1 -2493.125,E2 -2493.125} C_VEL
LIN {X 0,Y 566.95,Z 623.916,A -85,B 0,C 180,E1 -2494.451,E2 -2494.451} C_VEL
LIN {X 0,Y 566.872,Z 637.61,A -85,B 0,C 180,E1 -2494.774,E2 -2494.774} C_VEL
LIN {X 0,Y 566.688,Z 649.685,A -85,B 0,C 180,E1 -2495.207,E2 -2495.207} C_VEL
LIN {X 0,Y 566.585,Z 660.84,A -85,B 0,C 180,E1 -2495.74,E2 -2495.74} C_VEL
LIN {X 0,Y 566.48,Z 671.997,A -85,B 0,C 180,E1 -2496.415,E2 -2496.415} C_VEL
LIN {X 0,Y 566.329,Z 682.056,A -85,B 0,C 180,E1 -2497.182,E2 -2497.182} C_VEL
LIN {X 0,Y 566.208,Z 690.379,A -85,B 0,C 180,E1 -2497.947,E2 -2497.947} C_VEL
LIN {X 0,Y 566.094,Z 698.992,A -85,B 0,C 180,E1 -2498.898,E2 -2498.898} C_VEL
LIN {X 0,Y 566.021,Z 707.23,A -85,B 0,C 180,E1 -2500.035,E2 -2500.035} C_VEL
LIN {X 0,Y 565.973,Z 713.768,A -85,B 0,C 180,E1 -2501.165,E2 -2501.165} C_VEL
LIN {X 0,Y 565.908,Z 718.874,A -85,B 0,C 180,E1 -2502.286,E2 -2502.286} C_VEL
LIN {X 0,Y 565.884,Z 722.723,A -85,B 0,C 180,E1 -2503.403,E2 -2503.403} C_VEL
LIN {X 0,Y 565.836,Z 724.68,A -85,B 0,C 180,E1 -2504.142,E2 -2504.142} C_VEL
LIN {X 0,Y 565.815,Z 726.147,A -85,B 0,C 180,E1 -2504.88,E2 -2504.88} C_VEL
LIN {X 0,Y 565.867,Z 727.791,A -85,B 0,C 180,E1 -2506.351,E2 -2506.351} C_VEL
LIN {X 0,Y 565.845,Z 727.997,A -85,B 0,C 180,E1 -2507.082,E2 -2507.082} C_VEL
LIN {X 0,Y 565.868,Z 727.756,A -85,B 0,C 180,E1 -2507.811,E2 -2507.811} C_VEL
LIN {X 0,Y 565.896,Z 726.041,A -85,B 0,C 180,E1 -2509.264,E2 -2509.264} C_VEL
LIN {X 0,Y 565.887,Z 724.579,A -85,B 0,C 180,E1 -2509.987,E2 -2509.987} C_VEL
LIN {X 0,Y 565.898,Z 721.52,A -85,B 0,C 180,E1 -2511.07,E2 -2511.07} C_VEL
LIN {X 0,Y 565.953,Z 717.413,A -85,B 0,C 180,E1 -2512.149,E2 -2512.149} C_VEL
LIN {X 0,Y 566.007,Z 711.273,A -85,B 0,C 180,E1 -2513.392,E2 -2513.392} C_VEL
LIN {X 0,Y 566.011,Z 704.407,A -85,B 0,C 180,E1 -2514.478,E2 -2514.478} C_VEL
LIN {X 0,Y 566.16,Z 695.93,A -85,B 0,C 180,E1 -2515.551,E2 -2515.551} C_VEL
LIN {X 0,Y 566.237,Z 687.355,A -85,B 0,C 180,E1 -2516.442,E2 -2516.442} C_VEL
LIN {X 0,Y 566.401,Z 676.716,A -85,B 0,C 180,E1 -2517.333,E2 -2517.333} C_VEL
LIN {X 0,Y 566.525,Z 666.189,A -85,B 0,C 180,E1 -2518.045,E2 -2518.045} C_VEL
LIN {X 0,Y 566.645,Z 654.603,A -85,B 0,C 180,E1 -2518.668,E2 -2518.668} C_VEL
LIN {X 0,Y 566.824,Z 642.422,A -85,B 0,C 180,E1 -2519.157,E2 -2519.157} C_VEL
LIN {X 0,Y 566.901,Z 631.025,A -85,B 0,C 180,E1 -2519.49,E2 -2519.49} C_VEL
LIN {X 0,Y 566.999,Z 617.943,A -85,B 0,C 180,E1 -2519.734,E2 -2519.734} C_VEL
LIN {X 0,Y 567.021,Z 520.429,A -85,B 0,C 180,E1 -2520.977,E2 -2520.977} C_VEL
LIN {X 0,Y 566.381,Z 516.166,A -85,B 0,C 180,E1 -2521.067,E2 -2521.067} C_VEL
LIN {X 0,Y 566.399,Z 512.154,A -85,B 0,C 180,E1 -2521.6,E2 -2521.6} C_VEL
LIN {X 0,Y 566.601,Z 495.136,A -85,B 0,C 180,E1 -2524.09,E2 -2524.09} C_VEL
LIN {X 0,Y 566.81,Z 477.095,A -85,B 0,C 180,E1 -2526.765,E2 -2526.765} C_VEL
LIN {X 0,Y 567.08,Z 459.246,A -85,B 0,C 180,E1 -2529.452,E2 -2529.452} C_VEL
LIN {X 0,Y 566.201,Z 454.053,A -85,B 0,C 180,E1 -2530.301,E2 -2530.301} C_VEL
LIN {X 0,Y 566.185,Z 453.956,A -85,B 0,C 180,E1 -2532.182,E2 -2532.182} C_VEL
LIN {X 0,Y 566.189,Z 453.962,A -85,B 0,C 180,E1 -2535.11,E2 -2535.11} C_VEL
LIN {X 0,Y 566.193,Z 453.96,A -85,B 0,C 180,E1 -2537.332,E2 -2537.332} C_VEL
LIN {X 0,Y 566.205,Z 453.954,A -85,B 0,C 180,E1 -2539.581,E2 -2539.581} C_VEL
LIN {X 0,Y 566.193,Z 453.953,A -85,B 0,C 180,E1 -2541.863,E2 -2541.863} C_VEL
LIN {X 0,Y 566.192,Z 453.961,A -85,B 0,C 180,E1 -2545.022,E2 -2545.022} C_VEL
LIN {X 0,Y 566.214,Z 453.953,A -85,B 0,C 180,E1 -2547.339,E2 -2547.339} C_VEL
LIN {X 0,Y 566.205,Z 453.951,A -85,B 0,C 180,E1 -2549.769,E2 -2549.769} C_VEL
LIN {X 0,Y 566.212,Z 453.955,A -85,B 0,C 180,E1 -2552.43,E2 -2552.43} C_VEL
LIN {X 0,Y 566.19,Z 453.958,A -85,B 0,C 180,E1 -2554.989,E2 -2554.989} C_VEL
LIN {X 0,Y 566.204,Z 453.951,A -85,B 0,C 180,E1 -2557.461,E2 -2557.461} C_VEL
LIN {X 0,Y 566.215,Z 453.954,A -85,B 0,C 180,E1 -2560.199,E2 -2560.199} C_VEL
LIN {X 0,Y 566.207,Z 453.953,A -85,B 0,C 180,E1 -2563.054,E2 -2563.054} C_VEL
LIN {X 0,Y 566.201,Z 453.956,A -85,B 0,C 180,E1 -2566.049,E2 -2566.049} C_VEL
LIN {X 0,Y 566.211,Z 453.951,A -85,B 0,C 180,E1 -2569.214,E2 -2569.214} C_VEL
LIN {X 0,Y 566.189,Z 453.951,A -85,B 0,C 180,E1 -2571.636,E2 -2571.636} C_VEL
LIN {X 0,Y 566.15,Z 453.965,A -85,B 0,C 180,E1 -2574.306,E2 -2574.306} C_VEL
LIN {X 0,Y 566.209,Z 453.953,A -85,B 0,C 180,E1 -2576.896,E2 -2576.896} C_VEL
LIN {X 0,Y 566.181,Z 453.956,A -85,B 0,C 180,E1 -2579.406,E2 -2579.406} C_VEL
LIN {X 0,Y 566.208,Z 453.99,A -85,B 0,C 180,E1 -2582.56,E2 -2582.56} C_VEL
LIN {X 0,Y 566.276,Z 454.399,A -85,B 0,C 180,E1 -2582.663,E2 -2582.663} C_VEL
LIN {X 0,Y 567.95,Z 461.609,A -85,B 0,C 180,E1 -2583.545,E2 -2583.545} C_VEL
LIN {X 0,Y 567.801,Z 482.968,A -85,B 0,C 180,E1 -2585.891,E2 -2585.891} C_VEL
LIN {X 0,Y 567.404,Z 508.567,A -85,B 0,C 180,E1 -2588.787,E2 -2588.787} C_VEL
LIN {X 0,Y 566.979,Z 535.31,A -85,B 0,C 180,E1 -2591.76,E2 -2591.76} C_VEL
LIN {X 0,Y 566.667,Z 560.626,A -85,B 0,C 180,E1 -2594.534,E2 -2594.534} C_VEL
LIN {X 0,Y 566.554,Z 573.851,A -85,B 0,C 180,E1 -2595.955,E2 -2595.955} C_VEL
LIN {X 0,Y 567.209,Z 579.633,A -85,B 0,C 180,E1 -2596.063,E2 -2596.063} C_VEL
LIN {X 0,Y 566.964,Z 683.89,A -85,B 0,C 180,E1 -2597.402,E2 -2597.402} C_VEL
LIN {X 0,Y 566.879,Z 697.182,A -85,B 0,C 180,E1 -2597.718,E2 -2597.718} C_VEL
LIN {X 0,Y 566.762,Z 710.125,A -85,B 0,C 180,E1 -2598.179,E2 -2598.179} C_VEL
LIN {X 0,Y 566.607,Z 722.229,A -85,B 0,C 180,E1 -2598.769,E2 -2598.769} C_VEL
LIN {X 0,Y 566.421,Z 734.466,A -85,B 0,C 180,E1 -2599.544,E2 -2599.544} C_VEL
LIN {X 0,Y 566.298,Z 744.634,A -85,B 0,C 180,E1 -2600.354,E2 -2600.354} C_VEL
LIN {X 0,Y 566.163,Z 753.776,A -85,B 0,C 180,E1 -2601.252,E2 -2601.252} C_VEL
LIN {X 0,Y 566.082,Z 762.681,A -85,B 0,C 180,E1 -2602.329,E2 -2602.329} C_VEL
LIN {X 0,Y 565.969,Z 769.949,A -85,B 0,C 180,E1 -2603.421,E2 -2603.421} C_VEL
LIN {X 0,Y 566.004,Z 774.674,A -85,B 0,C 180,E1 -2604.298,E2 -2604.298} C_VEL
LIN {X 0,Y 565.933,Z 779.367,A -85,B 0,C 180,E1 -2605.369,E2 -2605.369} C_VEL
LIN {X 0,Y 565.927,Z 782.954,A -85,B 0,C 180,E1 -2606.439,E2 -2606.439} C_VEL
LIN {X 0,Y 565.878,Z 784.805,A -85,B 0,C 180,E1 -2607.151,E2 -2607.151} C_VEL
LIN {X 0,Y 565.845,Z 787.184,A -85,B 0,C 180,E1 -2608.575,E2 -2608.575} C_VEL
LIN {X 0,Y 565.839,Z 788,A -85,B 0,C 180,E1 -2609.999,E2 -2609.999} C_VEL
LIN {X 0,Y 565.845,Z 787.188,A -85,B 0,C 180,E1 -2611.422,E2 -2611.422} C_VEL
LIN {X 0,Y 565.877,Z 784.813,A -85,B 0,C 180,E1 -2612.846,E2 -2612.846} C_VEL
LIN {X 0,Y 565.926,Z 781.899,A -85,B 0,C 180,E1 -2613.915,E2 -2613.915} C_VEL
LIN {X 0,Y 565.878,Z 777.954,A -85,B 0,C 180,E1 -2614.986,E2 -2614.986} C_VEL
LIN {X 0,Y 566.002,Z 772.873,A -85,B 0,C 180,E1 -2616.057,E2 -2616.057} C_VEL
LIN {X 0,Y 566.039,Z 766.477,A -85,B 0,C 180,E1 -2617.131,E2 -2617.131} C_VEL
LIN {X 0,Y 566.133,Z 758.489,A -85,B 0,C 180,E1 -2618.206,E2 -2618.206} C_VEL
LIN {X 0,Y 566.228,Z 750.348,A -85,B 0,C 180,E1 -2619.104,E2 -2619.104} C_VEL
LIN {X 0,Y 566.342,Z 740.416,A -85,B 0,C 180,E1 -2620.004,E2 -2620.004} C_VEL
LIN {X 0,Y 566.543,Z 729.303,A -85,B 0,C 180,E1 -2620.806,E2 -2620.806} C_VEL
LIN {X 0,Y 566.658,Z 718.203,A -85,B 0,C 180,E1 -2621.444,E2 -2621.444} C_VEL
LIN {X 0,Y 566.743,Z 706.017,A -85,B 0,C 180,E1 -2621.987,E2 -2621.987} C_VEL
LIN {X 0,Y 566.909,Z 693.23,A -85,B 0,C 180,E1 -2622.392,E2 -2622.392} C_VEL
LIN {X 0,Y 566.999,Z 681.194,A -85,B 0,C 180,E1 -2622.64,E2 -2622.64} C_VEL
LIN {X 0,Y 567.102,Z 578.034,A -85,B 0,C 180,E1 -2623.96,E2 -2623.96} C_VEL
LIN {X 0,Y 566.555,Z 573.918,A -85,B 0,C 180,E1 -2624.043,E2 -2624.043} C_VEL
LIN {X 0,Y 566.832,Z 547.471,A -85,B 0,C 180,E1 -2626.917,E2 -2626.917} C_VEL
LIN {X 0,Y 567.167,Z 522.233,A -85,B 0,C 180,E1 -2629.714,E2 -2629.714} C_VEL
LIN {X 0,Y 567.575,Z 496.849,A -85,B 0,C 180,E1 -2632.571,E2 -2632.571} C_VEL
LIN {X 0,Y 567.816,Z 478.1,A -85,B 0,C 180,E1 -2634.69,E2 -2634.69} C_VEL
LIN {X 0,Y 567.999,Z 462.158,A -85,B 0,C 180,E1 -2636.45,E2 -2636.45} C_VEL
LIN {X 0,Y 566.188,Z 454.094,A -85,B 0,C 180,E1 -2637.464,E2 -2637.464} C_VEL
LIN {X 0,Y 566.165,Z 453.963,A -85,B 0,C 180,E1 -2639.769,E2 -2639.769} C_VEL
LIN {X 0,Y 566.196,Z 453.958,A -85,B 0,C 180,E1 -2642.428,E2 -2642.428} C_VEL
LIN {X 0,Y 566.159,Z 453.957,A -85,B 0,C 180,E1 -2644.986,E2 -2644.986} C_VEL
LIN {X 0,Y 566.178,Z 453.954,A -85,B 0,C 180,E1 -2647.46,E2 -2647.46} C_VEL
LIN {X 0,Y 566.197,Z 453.961,A -85,B 0,C 180,E1 -2650.198,E2 -2650.198} C_VEL
LIN {X 0,Y 566.178,Z 453.953,A -85,B 0,C 180,E1 -2653.054,E2 -2653.054} C_VEL
LIN {X 0,Y 566.183,Z 453.96,A -85,B 0,C 180,E1 -2656.048,E2 -2656.048} C_VEL
LIN {X 0,Y 566.193,Z 453.951,A -85,B 0,C 180,E1 -2659.214,E2 -2659.214} C_VEL
LIN {X 0,Y 566.169,Z 453.956,A -85,B 0,C 180,E1 -2661.635,E2 -2661.635} C_VEL
LIN {X 0,Y 566.138,Z 453.969,A -85,B 0,C 180,E1 -2664.306,E2 -2664.306} C_VEL
LIN {X 0,Y 566.208,Z 453.951,A -85,B 0,C 180,E1 -2666.897,E2 -2666.897} C_VEL
LIN {X 0,Y 566.163,Z 453.955,A -85,B 0,C 180,E1 -2669.406,E2 -2669.406} C_VEL
LIN {X 0,Y 566.181,Z 453.956,A -85,B 0,C 180,E1 -2671.855,E2 -2671.855} C_VEL
LIN {X 0,Y 566.192,Z 453.96,A -85,B 0,C 180,E1 -2674.25,E2 -2674.25} C_VEL
LIN {X 0,Y 566.159,Z 453.956,A -85,B 0,C 180,E1 -2677.367,E2 -2677.367} C_VEL
LIN {X 0,Y 566.196,Z 453.952,A -85,B 0,C 180,E1 -2679.662,E2 -2679.662} C_VEL
LIN {X 0,Y 566.183,Z 453.959,A -85,B 0,C 180,E1 -2682.668,E2 -2682.668} C_VEL
LIN {X 0,Y 566.201,Z 453.951,A -85,B 0,C 180,E1 -2685.626,E2 -2685.626} C_VEL
LIN {X 0,Y 566.263,Z 453.95,A -85,B 0,C 180,E1 -2688.653,E2 -2688.653} C_VEL
LIN {X 0,Y 566.191,Z 453.952,A -85,B 0,C 180,E1 -2691.433,E2 -2691.433} C_VEL
LIN {X 0,Y 566.241,Z 453.952,A -85,B 0,C 180,E1 -2694.301,E2 -2694.301} C_VEL
LIN {X 0,Y 566.256,Z 453.945,A -85,B 0,C 180,E1 -2697.866,E2 -2697.866} C_VEL
LIN {X 0,Y 566.298,Z 453.946,A -85,B 0,C 180,E1 -2700.711,E2 -2700.711} C_VEL
LIN {X 0,Y 566.17,Z 453.954,A -85,B 0,C 180,E1 -2703.558,E2 -2703.558} C_VEL
LIN {X 0,Y 566.241,Z 453.945,A -85,B 0,C 180,E1 -2705.698,E2 -2705.698} C_VEL
LIN {X 0,Y 566.234,Z 453.956,A -85,B 0,C 180,E1 -2708.565,E2 -2708.565} C_VEL
LIN {X 0,Y 566.237,Z 453.946,A -85,B 0,C 180,E1 -2711.454,E2 -2711.454} C_VEL
LIN {X 0,Y 566.219,Z 453.956,A -85,B 0,C 180,E1 -2714.507,E2 -2714.507} C_VEL
LIN {X 0,Y 566.187,Z 453.953,A -85,B 0,C 180,E1 -2717.332,E2 -2717.332} C_VEL
LIN {X 0,Y 566.206,Z 453.954,A -85,B 0,C 180,E1 -2720.337,E2 -2720.337} C_VEL
LIN {X 0,Y 566.175,Z 453.955,A -85,B 0,C 180,E1 -2723.404,E2 -2723.404} C_VEL
LIN {X 0,Y 566.2,Z 453.95,A -85,B 0,C 180,E1 -2725.749,E2 -2725.749} C_VEL
LIN {X 0,Y 566.2,Z 453.951,A -85,B 0,C 180,E1 -2727.501,E2 -2727.501} C_VEL
LIN {X 0,Y 565.523,Z 454.037,A -85,B 0,C 180,E1 -2728.095,E2 -2728.095} C_VEL
LIN {X 0,Y 562.653,Z 454.398,A -85,B 0,C 180,E1 -2729.058,E2 -2729.058} C_VEL
LIN {X 0,Y 560.239,Z 454.696,A -85,B 0,C 180,E1 -2729.834,E2 -2729.834} C_VEL
LIN {X 0,Y 559.211,Z 454.826,A -85,B 0,C 180,E1 -2730.433,E2 -2730.433} C_VEL
LIN {X 0,Y 559.133,Z 454.833,A -85,B 0,C 180,E1 -2730.635,E2 -2730.635} C_VEL
LIN {X 0,Y 559.165,Z 454.827,A -85,B 0,C 180,E1 -2733.574,E2 -2733.574} C_VEL
LIN {X 0,Y 559.155,Z 454.832,A -85,B 0,C 180,E1 -2736.449,E2 -2736.449} C_VEL
LIN {X 0,Y 559.166,Z 454.835,A -85,B 0,C 180,E1 -2738.934,E2 -2738.934} C_VEL
LIN {X 0,Y 559.181,Z 454.825,A -85,B 0,C 180,E1 -2741.768,E2 -2741.768} C_VEL
LIN {X 0,Y 559.129,Z 454.839,A -85,B 0,C 180,E1 -2744.74,E2 -2744.74} C_VEL
LIN {X 0,Y 559.158,Z 454.832,A -85,B 0,C 180,E1 -2747.258,E2 -2747.258} C_VEL
LIN {X 0,Y 559.177,Z 454.826,A -85,B 0,C 180,E1 -2750.136,E2 -2750.136} C_VEL
LIN {X 0,Y 559.136,Z 454.84,A -85,B 0,C 180,E1 -2752.893,E2 -2752.893} C_VEL
LIN {X 0,Y 559.158,Z 454.828,A -85,B 0,C 180,E1 -2756.052,E2 -2756.052} C_VEL
LIN {X 0,Y 559.157,Z 454.839,A -85,B 0,C 180,E1 -2758.983,E2 -2758.983} C_VEL
LIN {X 0,Y 559.185,Z 454.825,A -85,B 0,C 180,E1 -2762.29,E2 -2762.29} C_VEL
LIN {X 0,Y 559.173,Z 454.833,A -85,B 0,C 180,E1 -2764.814,E2 -2764.814} C_VEL
LIN {X 0,Y 559.136,Z 454.831,A -85,B 0,C 180,E1 -2767.848,E2 -2767.848} C_VEL
LIN {X 0,Y 559.192,Z 454.825,A -85,B 0,C 180,E1 -2770.494,E2 -2770.494} C_VEL
LIN {X 0,Y 559.18,Z 454.834,A -85,B 0,C 180,E1 -2773.199,E2 -2773.199} C_VEL
LIN {X 0,Y 559.17,Z 454.826,A -85,B 0,C 180,E1 -2776.185,E2 -2776.185} C_VEL
LIN {X 0,Y 559.193,Z 454.834,A -85,B 0,C 180,E1 -2779.135,E2 -2779.135} C_VEL
LIN {X 0,Y 559.204,Z 454.823,A -85,B 0,C 180,E1 -2782.055,E2 -2782.055} C_VEL
LIN {X 0,Y 559.255,Z 454.824,A -85,B 0,C 180,E1 -2784.955,E2 -2784.955} C_VEL
LIN {X 0,Y 559.254,Z 454.821,A -85,B 0,C 180,E1 -2787.841,E2 -2787.841} C_VEL
LIN {X 0,Y 559.281,Z 455.003,A -85,B 0,C 180,E1 -2790.114,E2 -2790.114} C_VEL
LIN {X 0,Y 559.486,Z 455.997,A -85,B 0,C 180,E1 -2790.226,E2 -2790.226} C_VEL
LIN {X 0,Y 560.226,Z 458.329,A -85,B 0,C 180,E1 -2790.286,E2 -2790.286} C_VEL
LIN {X 0,Y 560.099,Z 535.565,A -85,B 0,C 180,E1 -2791.304,E2 -2791.304} C_VEL
LIN {X 0,Y 559.941,Z 548.468,A -85,B 0,C 180,E1 -2791.619,E2 -2791.619} C_VEL
LIN {X 0,Y 559.832,Z 560.842,A -85,B 0,C 180,E1 -2792.07,E2 -2792.07} C_VEL
LIN {X 0,Y 559.709,Z 571.87,A -85,B 0,C 180,E1 -2792.61,E2 -2792.61} C_VEL
LIN {X 0,Y 559.509,Z 583.303,A -85,B 0,C 180,E1 -2793.332,E2 -2793.332} C_VEL
LIN {X 0,Y 559.332,Z 593.57,A -85,B 0,C 180,E1 -2794.144,E2 -2794.144} C_VEL
LIN {X 0,Y 559.173,Z 602.84,A -85,B 0,C 180,E1 -2795.049,E2 -2795.049} C_VEL
LIN {X 0,Y 559.051,Z 611.758,A -85,B 0,C 180,E1 -2796.135,E2 -2796.135} C_VEL
LIN {X 0,Y 558.981,Z 618.999,A -85,B 0,C 180,E1 -2797.224,E2 -2797.224} C_VEL
LIN {X 0,Y 558.875,Z 624.905,A -85,B 0,C 180,E1 -2798.316,E2 -2798.316} C_VEL
LIN {X 0,Y 558.803,Z 629.592,A -85,B 0,C 180,E1 -2799.411,E2 -2799.411} C_VEL
LIN {X 0,Y 558.817,Z 633.163,A -85,B 0,C 180,E1 -2800.508,E2 -2800.508} C_VEL
LIN {X 0,Y 558.772,Z 635.721,A -85,B 0,C 180,E1 -2801.611,E2 -2801.611} C_VEL
LIN {X 0,Y 558.771,Z 636.9,A -85,B 0,C 180,E1 -2802.347,E2 -2802.347} C_VEL
LIN {X 0,Y 558.743,Z 637.628,A -85,B 0,C 180,E1 -2803.087,E2 -2803.087} C_VEL
LIN {X 0,Y 558.758,Z 637.923,A -85,B 0,C 180,E1 -2804.421,E2 -2804.421} C_VEL
LIN {X 0,Y 558.709,Z 637.367,A -85,B 0,C 180,E1 -2805.318,E2 -2805.318} C_VEL
LIN {X 0,Y 558.73,Z 636.412,A -85,B 0,C 180,E1 -2806.066,E2 -2806.066} C_VEL
LIN {X 0,Y 558.768,Z 634.443,A -85,B 0,C 180,E1 -2807.08,E2 -2807.08} C_VEL
LIN {X 0,Y 558.814,Z 630.835,A -85,B 0,C 180,E1 -2808.327,E2 -2808.327} C_VEL
LIN {X 0,Y 558.885,Z 625.768,A -85,B 0,C 180,E1 -2809.591,E2 -2809.591} C_VEL
LIN {X 0,Y 558.929,Z 619.339,A -85,B 0,C 180,E1 -2810.808,E2 -2810.808} C_VEL
LIN {X 0,Y 559.048,Z 611.624,A -85,B 0,C 180,E1 -2811.975,E2 -2811.975} C_VEL
LIN {X 0,Y 559.165,Z 603.821,A -85,B 0,C 180,E1 -2812.933,E2 -2812.933} C_VEL
LIN {X 0,Y 559.339,Z 594.05,A -85,B 0,C 180,E1 -2813.906,E2 -2813.906} C_VEL
LIN {X 0,Y 559.47,Z 584.306,A -85,B 0,C 180,E1 -2814.689,E2 -2814.689} C_VEL
LIN {X 0,Y 559.681,Z 573.898,A -85,B 0,C 180,E1 -2815.364,E2 -2815.364} C_VEL
LIN {X 0,Y 559.839,Z 562.139,A -85,B 0,C 180,E1 -2815.965,E2 -2815.965} C_VEL
LIN {X 0,Y 559.982,Z 549.688,A -85,B 0,C 180,E1 -2816.434,E2 -2816.434} C_VEL
LIN {X 0,Y 560.07,Z 536.492,A -85,B 0,C 180,E1 -2816.769,E2 -2816.769} C_VEL
LIN {X 0,Y 560.149,Z 505.152,A -85,B 0,C 180,E1 -2817.2,E2 -2817.2} C_VEL
LIN {X 0,Y 560.161,Z 458.252,A -85,B 0,C 180,E1 -2817.808,E2 -2817.808} C_VEL
LIN {X 0,Y 559.365,Z 455.609,A -85,B 0,C 180,E1 -2817.892,E2 -2817.892} C_VEL
LIN {X 0,Y 559.196,Z 454.912,A -85,B 0,C 180,E1 -2818.014,E2 -2818.014} C_VEL
LIN {X 0,Y 559.159,Z 454.837,A -85,B 0,C 180,E1 -2821.02,E2 -2821.02} C_VEL
LIN {X 0,Y 559.16,Z 454.83,A -85,B 0,C 180,E1 -2823.949,E2 -2823.949} C_VEL
LIN {X 0,Y 559.144,Z 454.836,A -85,B 0,C 180,E1 -2827.109,E2 -2827.109} C_VEL
LIN {X 0,Y 559.163,Z 454.827,A -85,B 0,C 180,E1 -2829.942,E2 -2829.942} C_VEL
LIN {X 0,Y 559.162,Z 454.835,A -85,B 0,C 180,E1 -2832.745,E2 -2832.745} C_VEL
LIN {X 0,Y 559.152,Z 454.83,A -85,B 0,C 180,E1 -2835.762,E2 -2835.762} C_VEL
LIN {X 0,Y 559.166,Z 454.83,A -85,B 0,C 180,E1 -2838.23,E2 -2838.23} C_VEL
LIN {X 0,Y 559.176,Z 454.832,A -85,B 0,C 180,E1 -2841.193,E2 -2841.193} C_VEL
LIN {X 0,Y 559.212,Z 455.028,A -85,B 0,C 180,E1 -2843.735,E2 -2843.735} C_VEL
LIN {X 0,Y 560.116,Z 460.837,A -85,B 0,C 180,E1 -2844.646,E2 -2844.646} C_VEL
LIN {X 0,Y 559.881,Z 478.647,A -85,B 0,C 180,E1 -2847.333,E2 -2847.333} C_VEL
LIN {X 0,Y 559.563,Z 498.567,A -85,B 0,C 180,E1 -2850.306,E2 -2850.306} C_VEL
LIN {X 0,Y 559.387,Z 515.775,A -85,B 0,C 180,E1 -2852.816,E2 -2852.816} C_VEL
LIN {X 0,Y 559.816,Z 518.918,A -85,B 0,C 180,E1 -2852.911,E2 -2852.911} C_VEL
LIN {X 0,Y 560.33,Z 524.427,A -85,B 0,C 180,E1 -2852.995,E2 -2852.995} C_VEL
LIN {X 0,Y 560.038,Z 624.056,A -85,B 0,C 180,E1 -2854.296,E2 -2854.296} C_VEL
LIN {X 0,Y 559.952,Z 636.849,A -85,B 0,C 180,E1 -2854.597,E2 -2854.597} C_VEL
LIN {X 0,Y 559.754,Z 648.965,A -85,B 0,C 180,E1 -2855.028,E2 -2855.028} C_VEL
LIN {X 0,Y 559.653,Z 659.33,A -85,B 0,C 180,E1 -2855.518,E2 -2855.518} C_VEL
LIN {X 0,Y 559.491,Z 669.3,A -85,B 0,C 180,E1 -2856.103,E2 -2856.103} C_VEL
LIN {X 0,Y 559.324,Z 680.438,A -85,B 0,C 180,E1 -2856.918,E2 -2856.918} C_VEL
LIN {X 0,Y 559.194,Z 688.627,A -85,B 0,C 180,E1 -2857.655,E2 -2857.655} C_VEL
LIN {X 0,Y 559.096,Z 697.536,A -85,B 0,C 180,E1 -2858.621,E2 -2858.621} C_VEL
LIN {X 0,Y 558.951,Z 706.137,A -85,B 0,C 180,E1 -2859.771,E2 -2859.771} C_VEL
LIN {X 0,Y 558.913,Z 712.86,A -85,B 0,C 180,E1 -2860.917,E2 -2860.917} C_VEL
LIN {X 0,Y 558.828,Z 718.179,A -85,B 0,C 180,E1 -2862.054,E2 -2862.054} C_VEL
LIN {X 0,Y 558.819,Z 722.227,A -85,B 0,C 180,E1 -2863.187,E2 -2863.187} C_VEL
LIN {X 0,Y 558.756,Z 724.265,A -85,B 0,C 180,E1 -2863.936,E2 -2863.936} C_VEL
LIN {X 0,Y 558.722,Z 725.825,A -85,B 0,C 180,E1 -2864.684,E2 -2864.684} C_VEL
LIN {X 0,Y 558.764,Z 727.133,A -85,B 0,C 180,E1 -2865.581,E2 -2865.581} C_VEL
LIN {X 0,Y 558.746,Z 727.978,A -85,B 0,C 180,E1 -2866.915,E2 -2866.915} C_VEL
LIN {X 0,Y 558.774,Z 727.819,A -85,B 0,C 180,E1 -2867.654,E2 -2867.654} C_VEL
LIN {X 0,Y 558.797,Z 726.336,A -85,B 0,C 180,E1 -2869.126,E2 -2869.126} C_VEL
LIN {X 0,Y 558.784,Z 724.955,A -85,B 0,C 180,E1 -2869.859,E2 -2869.859} C_VEL
LIN {X 0,Y 558.808,Z 722.072,A -85,B 0,C 180,E1 -2870.955,E2 -2870.955} C_VEL
LIN {X 0,Y 558.871,Z 718.118,A -85,B 0,C 180,E1 -2872.049,E2 -2872.049} C_VEL
LIN {X 0,Y 558.91,Z 713.031,A -85,B 0,C 180,E1 -2873.14,E2 -2873.14} C_VEL
LIN {X 0,Y 558.97,Z 706.709,A -85,B 0,C 180,E1 -2874.227,E2 -2874.227} C_VEL
LIN {X 0,Y 559.041,Z 698.845,A -85,B 0,C 180,E1 -2875.313,E2 -2875.313} C_VEL
LIN {X 0,Y 559.174,Z 690.783,A -85,B 0,C 180,E1 -2876.217,E2 -2876.217} C_VEL
LIN {X 0,Y 559.272,Z 681.068,A -85,B 0,C 180,E1 -2877.119,E2 -2877.119} C_VEL
LIN {X 0,Y 559.498,Z 670.173,A -85,B 0,C 180,E1 -2877.931,E2 -2877.931} C_VEL
LIN {X 0,Y 559.587,Z 659.562,A -85,B 0,C 180,E1 -2878.561,E2 -2878.561} C_VEL
LIN {X 0,Y 559.817,Z 648.04,A -85,B 0,C 180,E1 -2879.101,E2 -2879.101} C_VEL
LIN {X 0,Y 559.953,Z 634.746,A -85,B 0,C 180,E1 -2879.551,E2 -2879.551} C_VEL
LIN {X 0,Y 560.037,Z 622.49,A -85,B 0,C 180,E1 -2879.821,E2 -2879.821} C_VEL
LIN {X 0,Y 560.215,Z 521.575,A -85,B 0,C 180,E1 -2881.135,E2 -2881.135} C_VEL
LIN {X 0,Y 559.354,Z 515.97,A -85,B 0,C 180,E1 -2881.26,E2 -2881.26} C_VEL
LIN {X 0,Y 559.562,Z 501.104,A -85,B 0,C 180,E1 -2883.421,E2 -2883.421} C_VEL
LIN {X 0,Y 559.831,Z 481.809,A -85,B 0,C 180,E1 -2886.307,E2 -2886.307} C_VEL
LIN {X 0,Y 560.137,Z 461.425,A -85,B 0,C 180,E1 -2889.388,E2 -2889.388} C_VEL
LIN {X 0,Y 559.492,Z 456.548,A -85,B 0,C 180,E1 -2890.129,E2 -2890.129} C_VEL
LIN {X 0,Y 559.184,Z 454.888,A -85,B 0,C 180,E1 -2890.409,E2 -2890.409} C_VEL
LIN {X 0,Y 559.142,Z 454.84,A -85,B 0,C 180,E1 -2893.076,E2 -2893.076} C_VEL
LIN {X 0,Y 559.139,Z 454.84,A -85,B 0,C 180,E1 -2895.305,E2 -2895.305} C_VEL
LIN {X 0,Y 559.137,Z 454.836,A -85,B 0,C 180,E1 -2897.558,E2 -2897.558} C_VEL
LIN {X 0,Y 559.169,Z 454.829,A -85,B 0,C 180,E1 -2899.838,E2 -2899.838} C_VEL
LIN {X 0,Y 559.141,Z 454.832,A -85,B 0,C 180,E1 -2902.153,E2 -2902.153} C_VEL
LIN {X 0,Y 559.151,Z 454.836,A -85,B 0,C 180,E1 -2905.179,E2 -2905.179} C_VEL
LIN {X 0,Y 559.154,Z 454.83,A -85,B 0,C 180,E1 -2907.714,E2 -2907.714} C_VEL
LIN {X 0,Y 559.158,Z 454.831,A -85,B 0,C 180,E1 -2910.183,E2 -2910.183} C_VEL
LIN {X 0,Y 559.165,Z 454.837,A -85,B 0,C 180,E1 -2912.715,E2 -2912.715} C_VEL
LIN {X 0,Y 559.136,Z 454.833,A -85,B 0,C 180,E1 -2915.324,E2 -2915.324} C_VEL
LIN {X 0,Y 559.14,Z 454.833,A -85,B 0,C 180,E1 -2918.017,E2 -2918.017} C_VEL
LIN {X 0,Y 559.163,Z 454.834,A -85,B 0,C 180,E1 -2920.812,E2 -2920.812} C_VEL
LIN {X 0,Y 559.145,Z 454.832,A -85,B 0,C 180,E1 -2923.734,E2 -2923.734} C_VEL
LIN {X 0,Y 559.152,Z 454.834,A -85,B 0,C 180,E1 -2926.803,E2 -2926.803} C_VEL
LIN {X 0,Y 559.163,Z 454.829,A -85,B 0,C 180,E1 -2929.187,E2 -2929.187} C_VEL
LIN {X 0,Y 559.136,Z 454.833,A -85,B 0,C 180,E1 -2931.982,E2 -2931.982} C_VEL
LIN {X 0,Y 559.13,Z 454.833,A -85,B 0,C 180,E1 -2934.788,E2 -2934.788} C_VEL
LIN {X 0,Y 559.16,Z 454.831,A -85,B 0,C 180,E1 -2937.364,E2 -2937.364} C_VEL
LIN {X 0,Y 559.147,Z 454.839,A -85,B 0,C 180,E1 -2940.143,E2 -2940.143} C_VEL
LIN {X 0,Y 559.167,Z 454.967,A -85,B 0,C 180,E1 -2942.434,E2 -2942.434} C_VEL
LIN {X 0,Y 560.985,Z 462.547,A -85,B 0,C 180,E1 -2943.392,E2 -2943.392} C_VEL
LIN {X 0,Y 560.874,Z 478.48,A -85,B 0,C 180,E1 -2945.179,E2 -2945.179} C_VEL
LIN {X 0,Y 560.678,Z 501.552,A -85,B 0,C 180,E1 -2947.716,E2 -2947.716} C_VEL
LIN {X 0,Y 560.23,Z 525.803,A -85,B 0,C 180,E1 -2950.461,E2 -2950.461} C_VEL
LIN {X 0,Y 559.861,Z 552.188,A -85,B 0,C 180,E1 -2953.405,E2 -2953.405} C_VEL
LIN {X 0,Y 559.599,Z 573.855,A -85,B 0,C 180,E1 -2955.777,E2 -2955.777} C_VEL
LIN {X 0,Y 560.325,Z 581.422,A -85,B 0,C 180,E1 -2955.911,E2 -2955.911} C_VEL
LIN {X 0,Y 560.059,Z 683.89,A -85,B 0,C 180,E1 -2957.244,E2 -2957.244} C_VEL
LIN {X 0,Y 559.938,Z 697.181,A -85,B 0,C 180,E1 -2957.564,E2 -2957.564} C_VEL
LIN {X 0,Y 559.794,Z 710.126,A -85,B 0,C 180,E1 -2958.03,E2 -2958.03} C_VEL
LIN {X 0,Y 559.636,Z 722.829,A -85,B 0,C 180,E1 -2958.662,E2 -2958.662} C_VEL
LIN {X 0,Y 559.437,Z 734.468,A -85,B 0,C 180,E1 -2959.412,E2 -2959.412} C_VEL
LIN {X 0,Y 559.294,Z 744.634,A -85,B 0,C 180,E1 -2960.232,E2 -2960.232} C_VEL
LIN {X 0,Y 559.133,Z 753.776,A -85,B 0,C 180,E1 -2961.141,E2 -2961.141} C_VEL
LIN {X 0,Y 559.011,Z 762.681,A -85,B 0,C 180,E1 -2962.231,E2 -2962.231} C_VEL
LIN {X 0,Y 558.926,Z 768.734,A -85,B 0,C 180,E1 -2963.139,E2 -2963.139} C_VEL
LIN {X 0,Y 558.936,Z 774.674,A -85,B 0,C 180,E1 -2964.226,E2 -2964.226} C_VEL
LIN {X 0,Y 558.827,Z 779.368,A -85,B 0,C 180,E1 -2965.31,E2 -2965.31} C_VEL
LIN {X 0,Y 558.836,Z 782.954,A -85,B 0,C 180,E1 -2966.394,E2 -2966.394} C_VEL
LIN {X 0,Y 558.799,Z 784.805,A -85,B 0,C 180,E1 -2967.115,E2 -2967.115} C_VEL
LIN {X 0,Y 558.745,Z 787.184,A -85,B 0,C 180,E1 -2968.557,E2 -2968.557} C_VEL
LIN {X 0,Y 558.74,Z 788,A -85,B 0,C 180,E1 -2969.999,E2 -2969.999} C_VEL
LIN {X 0,Y 558.745,Z 787.187,A -85,B 0,C 180,E1 -2971.44,E2 -2971.44} C_VEL
LIN {X 0,Y 558.799,Z 784.813,A -85,B 0,C 180,E1 -2972.882,E2 -2972.882} C_VEL
LIN {X 0,Y 558.844,Z 781.899,A -85,B 0,C 180,E1 -2973.965,E2 -2973.965} C_VEL
LIN {X 0,Y 558.798,Z 777.954,A -85,B 0,C 180,E1 -2975.05,E2 -2975.05} C_VEL
LIN {X 0,Y 558.918,Z 772.873,A -85,B 0,C 180,E1 -2976.134,E2 -2976.134} C_VEL
LIN {X 0,Y 558.976,Z 766.477,A -85,B 0,C 180,E1 -2977.222,E2 -2977.222} C_VEL
LIN {X 0,Y 559.098,Z 758.488,A -85,B 0,C 180,E1 -2978.31,E2 -2978.31} C_VEL
LIN {X 0,Y 559.184,Z 750.348,A -85,B 0,C 180,E1 -2979.22,E2 -2979.22} C_VEL
LIN {X 0,Y 559.342,Z 740.416,A -85,B 0,C 180,E1 -2980.13,E2 -2980.13} C_VEL
LIN {X 0,Y 559.557,Z 729.384,A -85,B 0,C 180,E1 -2980.938,E2 -2980.938} C_VEL
LIN {X 0,Y 559.701,Z 717.168,A -85,B 0,C 180,E1 -2981.642,E2 -2981.642} C_VEL
LIN {X 0,Y 559.831,Z 704.805,A -85,B 0,C 180,E1 -2982.183,E2 -2982.183} C_VEL
LIN {X 0,Y 559.98,Z 691.4,A -85,B 0,C 180,E1 -2982.594,E2 -2982.594} C_VEL
LIN {X 0,Y 560.103,Z 678.178,A -85,B 0,C 180,E1 -2982.845,E2 -2982.845} C_VEL
LIN {X 0,Y 560.179,Z 578.485,A -85,B 0,C 180,E1 -2984.131,E2 -2984.131} C_VEL
LIN {X 0,Y 559.597,Z 573.924,A -85,B 0,C 180,E1 -2984.221,E2 -2984.221} C_VEL
LIN {X 0,Y 559.9,Z 546.775,A -85,B 0,C 180,E1 -2987.211,E2 -2987.211} C_VEL
LIN {X 0,Y 560.344,Z 520.386,A -85,B 0,C 180,E1 -2990.175,E2 -2990.175} C_VEL
LIN {X 0,Y 560.754,Z 494.917,A -85,B 0,C 180,E1 -2993.056,E2 -2993.056} C_VEL
LIN {X 0,Y 561.054,Z 468.39,A -85,B 0,C 180,E1 -2996.002,E2 -2996.002} C_VEL
LIN {X 0,Y 561.067,Z 463.136,A -85,B 0,C 180,E1 -2996.602,E2 -2996.602} C_VEL
LIN {X 0,Y 559.177,Z 454.991,A -85,B 0,C 180,E1 -2997.64,E2 -2997.64} C_VEL
LIN {X 0,Y 559.131,Z 454.841,A -85,B 0,C 180,E1 -3000.182,E2 -3000.182} C_VEL
LIN {X 0,Y 559.146,Z 454.833,A -85,B 0,C 180,E1 -3002.714,E2 -3002.714} C_VEL
LIN {X 0,Y 559.109,Z 454.835,A -85,B 0,C 180,E1 -3005.324,E2 -3005.324} C_VEL
LIN {X 0,Y 559.117,Z 454.841,A -85,B 0,C 180,E1 -3008.017,E2 -3008.017} C_VEL
LIN {X 0,Y 559.119,Z 454.834,A -85,B 0,C 180,E1 -3010.814,E2 -3010.814} C_VEL
LIN {X 0,Y 559.122,Z 454.832,A -85,B 0,C 180,E1 -3013.193,E2 -3013.193} C_VEL
LIN {X 0,Y 559.125,Z 454.842,A -85,B 0,C 180,E1 -3016.264,E2 -3016.264} C_VEL
LIN {X 0,Y 559.144,Z 454.829,A -85,B 0,C 180,E1 -3019.186,E2 -3019.186} C_VEL
LIN {X 0,Y 559.117,Z 454.838,A -85,B 0,C 180,E1 -3021.981,E2 -3021.981} C_VEL
LIN {X 0,Y 559.117,Z 454.836,A -85,B 0,C 180,E1 -3024.787,E2 -3024.787} C_VEL
LIN {X 0,Y 559.144,Z 454.829,A -85,B 0,C 180,E1 -3027.363,E2 -3027.363} C_VEL
LIN {X 0,Y 559.131,Z 454.838,A -85,B 0,C 180,E1 -3030.143,E2 -3030.143} C_VEL
LIN {X 0,Y 559.153,Z 454.829,A -85,B 0,C 180,E1 -3033.173,E2 -3033.173} C_VEL
LIN {X 0,Y 559.112,Z 454.834,A -85,B 0,C 180,E1 -3035.493,E2 -3035.493} C_VEL
LIN {X 0,Y 559.157,Z 454.834,A -85,B 0,C 180,E1 -3038.623,E2 -3038.623} C_VEL
LIN {X 0,Y 559.146,Z 454.832,A -85,B 0,C 180,E1 -3040.925,E2 -3040.925} C_VEL
LIN {X 0,Y 559.146,Z 454.832,A -85,B 0,C 180,E1 -3043.947,E2 -3043.947} C_VEL
LIN {X 0,Y 559.146,Z 454.835,A -85,B 0,C 180,E1 -3046.183,E2 -3046.183} C_VEL
LIN {X 0,Y 559.201,Z 454.824,A -85,B 0,C 180,E1 -3049.133,E2 -3049.133} C_VEL
LIN {X 0,Y 559.186,Z 454.828,A -85,B 0,C 180,E1 -3052.053,E2 -3052.053} C_VEL
LIN {X 0,Y 559.236,Z 454.821,A -85,B 0,C 180,E1 -3054.953,E2 -3054.953} C_VEL
LIN {X 0,Y 559.229,Z 454.82,A -85,B 0,C 180,E1 -3057.839,E2 -3057.839} C_VEL
LIN {X 0,Y 559.267,Z 454.822,A -85,B 0,C 180,E1 -3060.72,E2 -3060.72} C_VEL
LIN {X 0,Y 559.233,Z 454.823,A -85,B 0,C 180,E1 -3062.881,E2 -3062.881} C_VEL
LIN {X 0,Y 559.21,Z 454.822,A -85,B 0,C 180,E1 -3065.77,E2 -3065.77} C_VEL
LIN {X 0,Y 559.189,Z 454.833,A -85,B 0,C 180,E1 -3068.674,E2 -3068.674} C_VEL
LIN {X 0,Y 559.195,Z 454.823,A -85,B 0,C 180,E1 -3071.6,E2 -3071.6} C_VEL
LIN {X 0,Y 559.185,Z 454.834,A -85,B 0,C 180,E1 -3074.596,E2 -3074.596} C_VEL
LIN {X 0,Y 559.146,Z 454.829,A -85,B 0,C 180,E1 -3077.557,E2 -3077.557} C_VEL
LIN {X 0,Y 559.161,Z 454.828,A -85,B 0,C 180,E1 -3079.837,E2 -3079.837} C_VEL
LIN {X 0,Y 559.129,Z 454.833,A -85,B 0,C 180,E1 -3082.153,E2 -3082.153} C_VEL
LIN {X 0,Y 559.165,Z 454.83,A -85,B 0,C 180,E1 -3085.188,E2 -3085.188} C_VEL
LIN {X 0,Y 559.18,Z 454.825,A -85,B 0,C 180,E1 -3087.712,E2 -3087.712} C_VEL
LIN {X 0,Y 559.133,Z 454.833,A -85,B 0,C 180,E1 -3090.635,E2 -3090.635} C_VEL
LIN {X 0,Y 558.475,Z 454.918,A -85,B 0,C 180,E1 -3091.237,E2 -3091.237} C_VEL
LIN {X 0,Y 555.615,Z 455.273,A -85,B 0,C 180,E1 -3092.213,E2 -3092.213} C_VEL
LIN {X 0,Y 553.203,Z 455.576,A -85,B 0,C 180,E1 -3092.999,E2 -3092.999} C_VEL
LIN {X 0,Y 552.185,Z 455.697,A -85,B 0,C 180,E1 -3093.606,E2 -3093.606} C_VEL
LIN {X 0,Y 552.111,Z 455.706,A -85,B 0,C 180,E1 -3093.811,E2 -3093.811} C_VEL
LIN {X 0,Y 552.099,Z 455.716,A -85,B 0,C 180,E1 -3096.747,E2 -3096.747} C_VEL
LIN {X 0,Y 552.122,Z 455.705,A -85,B 0,C 180,E1 -3099.527,E2 -3099.527} C_VEL
LIN {X 0,Y 552.119,Z 455.708,A -85,B 0,C 180,E1 -3102.426,E2 -3102.426} C_VEL
LIN {X 0,Y 552.089,Z 455.709,A -85,B 0,C 180,E1 -3105.564,E2 -3105.564} C_VEL
LIN {X 0,Y 552.161,Z 455.706,A -85,B 0,C 180,E1 -3108.673,E2 -3108.673} C_VEL
LIN {X 0,Y 552.111,Z 455.708,A -85,B 0,C 180,E1 -3111.412,E2 -3111.412} C_VEL
LIN {X 0,Y 552.094,Z 455.708,A -85,B 0,C 180,E1 -3114.159,E2 -3114.159} C_VEL
LIN {X 0,Y 552.115,Z 455.713,A -85,B 0,C 180,E1 -3116.816,E2 -3116.816} C_VEL
LIN {X 0,Y 552.101,Z 455.711,A -85,B 0,C 180,E1 -3119.392,E2 -3119.392} C_VEL
LIN {X 0,Y 552.119,Z 455.705,A -85,B 0,C 180,E1 -3121.904,E2 -3121.904} C_VEL
LIN {X 0,Y 552.149,Z 455.705,A -85,B 0,C 180,E1 -3124.651,E2 -3124.651} C_VEL
LIN {X 0,Y 552.09,Z 455.711,A -85,B 0,C 180,E1 -3127.55,E2 -3127.55} C_VEL
LIN {X 0,Y 552.144,Z 455.702,A -85,B 0,C 180,E1 -3130.375,E2 -3130.375} C_VEL
LIN {X 0,Y 552.152,Z 455.709,A -85,B 0,C 180,E1 -3132.979,E2 -3132.979} C_VEL
LIN {X 0,Y 552.133,Z 455.703,A -85,B 0,C 180,E1 -3136.006,E2 -3136.006} C_VEL
LIN {X 0,Y 552.16,Z 455.707,A -85,B 0,C 180,E1 -3138.995,E2 -3138.995} C_VEL
LIN {X 0,Y 552.158,Z 455.702,A -85,B 0,C 180,E1 -3141.953,E2 -3141.953} C_VEL
LIN {X 0,Y 552.23,Z 455.698,A -85,B 0,C 180,E1 -3144.89,E2 -3144.89} C_VEL
LIN {X 0,Y 552.225,Z 455.697,A -85,B 0,C 180,E1 -3147.813,E2 -3147.813} C_VEL
LIN {X 0,Y 552.25,Z 455.809,A -85,B 0,C 180,E1 -3149.91,E2 -3149.91} C_VEL
LIN {X 0,Y 552.468,Z 456.892,A -85,B 0,C 180,E1 -3150.047,E2 -3150.047} C_VEL
LIN {X 0,Y 553.339,Z 459.559,A -85,B 0,C 180,E1 -3150.115,E2 -3150.115} C_VEL
LIN {X 0,Y 553.231,Z 536.244,A -85,B 0,C 180,E1 -3151.139,E2 -3151.139} C_VEL
LIN {X 0,Y 553.086,Z 549.221,A -85,B 0,C 180,E1 -3151.457,E2 -3151.457} C_VEL
LIN {X 0,Y 552.944,Z 561.663,A -85,B 0,C 180,E1 -3151.913,E2 -3151.913} C_VEL
LIN {X 0,Y 552.81,Z 572.733,A -85,B 0,C 180,E1 -3152.46,E2 -3152.46} C_VEL
LIN {X 0,Y 552.612,Z 584.178,A -85,B 0,C 180,E1 -3153.191,E2 -3153.191} C_VEL
LIN {X 0,Y 552.422,Z 594.46,A -85,B 0,C 180,E1 -3154.014,E2 -3154.014} C_VEL
LIN {X 0,Y 552.227,Z 603.753,A -85,B 0,C 180,E1 -3154.929,E2 -3154.929} C_VEL
LIN {X 0,Y 552.084,Z 612.592,A -85,B 0,C 180,E1 -3156.017,E2 -3156.017} C_VEL
LIN {X 0,Y 552.004,Z 619.884,A -85,B 0,C 180,E1 -3157.132,E2 -3157.132} C_VEL
LIN {X 0,Y 551.862,Z 626.533,A -85,B 0,C 180,E1 -3158.423,E2 -3158.423} C_VEL
LIN {X 0,Y 551.77,Z 630.92,A -85,B 0,C 180,E1 -3159.532,E2 -3159.532} C_VEL
LIN {X 0,Y 551.761,Z 633.228,A -85,B 0,C 180,E1 -3160.273,E2 -3160.273} C_VEL
LIN {X 0,Y 551.725,Z 635.591,A -85,B 0,C 180,E1 -3161.235,E2 -3161.235} C_VEL
LIN {X 0,Y 551.697,Z 637.602,A -85,B 0,C 180,E1 -3162.508,E2 -3162.508} C_VEL
LIN {X 0,Y 551.672,Z 638.48,A -85,B 0,C 180,E1 -3164.009,E2 -3164.009} C_VEL
LIN {X 0,Y 551.645,Z 638.285,A -85,B 0,C 180,E1 -3164.763,E2 -3164.763} C_VEL
LIN {X 0,Y 551.647,Z 637.676,A -85,B 0,C 180,E1 -3165.519,E2 -3165.519} C_VEL
LIN {X 0,Y 551.67,Z 636.667,A -85,B 0,C 180,E1 -3166.277,E2 -3166.277} C_VEL
LIN {X 0,Y 551.712,Z 634.883,A -85,B 0,C 180,E1 -3167.18,E2 -3167.18} C_VEL
LIN {X 0,Y 551.766,Z 630.899,A -85,B 0,C 180,E1 -3168.569,E2 -3168.569} C_VEL
LIN {X 0,Y 551.87,Z 626.222,A -85,B 0,C 180,E1 -3169.744,E2 -3169.744} C_VEL
LIN {X 0,Y 551.969,Z 620.343,A -85,B 0,C 180,E1 -3170.887,E2 -3170.887} C_VEL
LIN {X 0,Y 552.083,Z 612.739,A -85,B 0,C 180,E1 -3172.058,E2 -3172.058} C_VEL
LIN {X 0,Y 552.22,Z 604.864,A -85,B 0,C 180,E1 -3173.04,E2 -3173.04} C_VEL
LIN {X 0,Y 552.42,Z 595.108,A -85,B 0,C 180,E1 -3174.025,E2 -3174.025} C_VEL
LIN {X 0,Y 552.608,Z 584.165,A -85,B 0,C 180,E1 -3174.905,E2 -3174.905} C_VEL
LIN {X 0,Y 552.853,Z 573.135,A -85,B 0,C 180,E1 -3175.609,E2 -3175.609} C_VEL
LIN {X 0,Y 552.973,Z 562.133,A -85,B 0,C 180,E1 -3176.16,E2 -3176.16} C_VEL
LIN {X 0,Y 553.102,Z 549.189,A -85,B 0,C 180,E1 -3176.636,E2 -3176.636} C_VEL
LIN {X 0,Y 553.218,Z 535.878,A -85,B 0,C 180,E1 -3176.961,E2 -3176.961} C_VEL
LIN {X 0,Y 553.357,Z 459.769,A -85,B 0,C 180,E1 -3177.973,E2 -3177.973} C_VEL
LIN {X 0,Y 552.307,Z 456.543,A -85,B 0,C 180,E1 -3178.071,E2 -3178.071} C_VEL
LIN {X 0,Y 552.153,Z 455.784,A -85,B 0,C 180,E1 -3178.21,E2 -3178.21} C_VEL
LIN {X 0,Y 552.106,Z 455.715,A -85,B 0,C 180,E1 -3180.61,E2 -3180.61} C_VEL
LIN {X 0,Y 552.11,Z 455.713,A -85,B 0,C 180,E1 -3183.187,E2 -3183.187} C_VEL
LIN {X 0,Y 552.089,Z 455.71,A -85,B 0,C 180,E1 -3185.845,E2 -3185.845} C_VEL
LIN {X 0,Y 552.119,Z 455.712,A -85,B 0,C 180,E1 -3188.59,E2 -3188.59} C_VEL
LIN {X 0,Y 552.124,Z 455.706,A -85,B 0,C 180,E1 -3191.447,E2 -3191.447} C_VEL
LIN {X 0,Y 552.093,Z 455.714,A -85,B 0,C 180,E1 -3194.532,E2 -3194.532} C_VEL
LIN {X 0,Y 552.134,Z 455.705,A -85,B 0,C 180,E1 -3197.585,E2 -3197.585} C_VEL
LIN {X 0,Y 552.132,Z 455.71,A -85,B 0,C 180,E1 -3200.473,E2 -3200.473} C_VEL
LIN {X 0,Y 552.152,Z 455.868,A -85,B 0,C 180,E1 -3203.583,E2 -3203.583} C_VEL
LIN {X 0,Y 553.093,Z 461.057,A -85,B 0,C 180,E1 -3204.414,E2 -3204.414} C_VEL
LIN {X 0,Y 552.948,Z 475.79,A -85,B 0,C 180,E1 -3206.653,E2 -3206.653} C_VEL
LIN {X 0,Y 552.65,Z 494.158,A -85,B 0,C 180,E1 -3209.425,E2 -3209.425} C_VEL
LIN {X 0,Y 552.366,Z 512.187,A -85,B 0,C 180,E1 -3212.123,E2 -3212.123} C_VEL
LIN {X 0,Y 552.386,Z 515.987,A -85,B 0,C 180,E1 -3212.648,E2 -3212.648} C_VEL
LIN {X 0,Y 553.427,Z 522.876,A -85,B 0,C 180,E1 -3212.796,E2 -3212.796} C_VEL
LIN {X 0,Y 553.127,Z 623.649,A -85,B 0,C 180,E1 -3214.128,E2 -3214.128} C_VEL
LIN {X 0,Y 553.025,Z 636.905,A -85,B 0,C 180,E1 -3214.44,E2 -3214.44} C_VEL
LIN {X 0,Y 552.799,Z 649.499,A -85,B 0,C 180,E1 -3214.899,E2 -3214.899} C_VEL
LIN {X 0,Y 552.698,Z 659.67,A -85,B 0,C 180,E1 -3215.39,E2 -3215.39} C_VEL
LIN {X 0,Y 552.492,Z 669.569,A -85,B 0,C 180,E1 -3215.98,E2 -3215.98} C_VEL
LIN {X 0,Y 552.293,Z 681.325,A -85,B 0,C 180,E1 -3216.866,E2 -3216.866} C_VEL
LIN {X 0,Y 552.147,Z 690.714,A -85,B 0,C 180,E1 -3217.749,E2 -3217.749} C_VEL
LIN {X 0,Y 552.015,Z 699.286,A -85,B 0,C 180,E1 -3218.725,E2 -3218.725} C_VEL
LIN {X 0,Y 551.879,Z 707.435,A -85,B 0,C 180,E1 -3219.89,E2 -3219.89} C_VEL
LIN {X 0,Y 551.849,Z 711.949,A -85,B 0,C 180,E1 -3220.664,E2 -3220.664} C_VEL
LIN {X 0,Y 551.737,Z 717.43,A -85,B 0,C 180,E1 -3221.816,E2 -3221.816} C_VEL
LIN {X 0,Y 551.744,Z 721.676,A -85,B 0,C 180,E1 -3222.964,E2 -3222.964} C_VEL
LIN {X 0,Y 551.679,Z 723.816,A -85,B 0,C 180,E1 -3223.724,E2 -3223.724} C_VEL
LIN {X 0,Y 551.623,Z 725.501,A -85,B 0,C 180,E1 -3224.482,E2 -3224.482} C_VEL
LIN {X 0,Y 551.654,Z 727.084,A -85,B 0,C 180,E1 -3225.522,E2 -3225.522} C_VEL
LIN {X 0,Y 551.659,Z 727.93,A -85,B 0,C 180,E1 -3226.744,E2 -3226.744} C_VEL
LIN {X 0,Y 551.675,Z 727.441,A -85,B 0,C 180,E1 -3228.239,E2 -3228.239} C_VEL
LIN {X 0,Y 551.705,Z 726.592,A -85,B 0,C 180,E1 -3228.984,E2 -3228.984} C_VEL
LIN {X 0,Y 551.681,Z 725.281,A -85,B 0,C 180,E1 -3229.727,E2 -3229.727} C_VEL
LIN {X 0,Y 551.701,Z 722.563,A -85,B 0,C 180,E1 -3230.838,E2 -3230.838} C_VEL
LIN {X 0,Y 551.767,Z 718.8,A -85,B 0,C 180,E1 -3231.946,E2 -3231.946} C_VEL
LIN {X 0,Y 551.827,Z 713.884,A -85,B 0,C 180,E1 -3233.051,E2 -3233.051} C_VEL
LIN {X 0,Y 551.905,Z 707.723,A -85,B 0,C 180,E1 -3234.153,E2 -3234.153} C_VEL
LIN {X 0,Y 551.975,Z 700.167,A -85,B 0,C 180,E1 -3235.253,E2 -3235.253} C_VEL
LIN {X 0,Y 552.08,Z 692.401,A -85,B 0,C 180,E1 -3236.168,E2 -3236.168} C_VEL
LIN {X 0,Y 552.235,Z 682.949,A -85,B 0,C 180,E1 -3237.082,E2 -3237.082} C_VEL
LIN {X 0,Y 552.472,Z 672.597,A -85,B 0,C 180,E1 -3237.904,E2 -3237.904} C_VEL
LIN {X 0,Y 552.607,Z 660.932,A -85,B 0,C 180,E1 -3238.634,E2 -3238.634} C_VEL
LIN {X 0,Y 552.824,Z 650.757,A -85,B 0,C 180,E1 -3239.135,E2 -3239.135} C_VEL
LIN {X 0,Y 553,Z 638.76,A -85,B 0,C 180,E1 -3239.591,E2 -3239.591} C_VEL
LIN {X 0,Y 553.115,Z 625.406,A -85,B 0,C 180,E1 -3239.932,E2 -3239.932} C_VEL
LIN {X 0,Y 553.245,Z 594.261,A -85,B 0,C 180,E1 -3240.364,E2 -3240.364} C_VEL
LIN {X 0,Y 553.271,Z 522.114,A -85,B 0,C 180,E1 -3241.308,E2 -3241.308} C_VEL
LIN {X 0,Y 552.38,Z 516.114,A -85,B 0,C 180,E1 -3241.436,E2 -3241.436} C_VEL
LIN {X 0,Y 552.462,Z 510.74,A -85,B 0,C 180,E1 -3242.187,E2 -3242.187} C_VEL
LIN {X 0,Y 552.632,Z 492.567,A -85,B 0,C 180,E1 -3244.925,E2 -3244.925} C_VEL
LIN {X 0,Y 552.919,Z 477.702,A -85,B 0,C 180,E1 -3247.172,E2 -3247.172} C_VEL
LIN {X 0,Y 553.103,Z 461.077,A -85,B 0,C 180,E1 -3249.693,E2 -3249.693} C_VEL
LIN {X 0,Y 552.157,Z 455.78,A -85,B 0,C 180,E1 -3250.52,E2 -3250.52} C_VEL
LIN {X 0,Y 552.105,Z 455.717,A -85,B 0,C 180,E1 -3253.246,E2 -3253.246} C_VEL
LIN {X 0,Y 552.099,Z 455.714,A -85,B 0,C 180,E1 -3255.505,E2 -3255.505} C_VEL
LIN {X 0,Y 552.095,Z 455.711,A -85,B 0,C 180,E1 -3257.789,E2 -3257.789} C_VEL
LIN {X 0,Y 552.13,Z 455.705,A -85,B 0,C 180,E1 -3260.102,E2 -3260.102} C_VEL
LIN {X 0,Y 552.093,Z 455.712,A -85,B 0,C 180,E1 -3262.451,E2 -3262.451} C_VEL
LIN {X 0,Y 552.115,Z 455.71,A -85,B 0,C 180,E1 -3265.339,E2 -3265.339} C_VEL
LIN {X 0,Y 552.1,Z 455.709,A -85,B 0,C 180,E1 -3268.099,E2 -3268.099} C_VEL
LIN {X 0,Y 552.108,Z 455.714,A -85,B 0,C 180,E1 -3270.609,E2 -3270.609} C_VEL
LIN {X 0,Y 552.124,Z 455.708,A -85,B 0,C 180,E1 -3273.186,E2 -3273.186} C_VEL
LIN {X 0,Y 552.094,Z 455.709,A -85,B 0,C 180,E1 -3275.843,E2 -3275.843} C_VEL
LIN {X 0,Y 552.129,Z 455.708,A -85,B 0,C 180,E1 -3279.061,E2 -3279.061} C_VEL
LIN {X 0,Y 552.128,Z 455.705,A -85,B 0,C 180,E1 -3281.446,E2 -3281.446} C_VEL
LIN {X 0,Y 552.097,Z 455.717,A -85,B 0,C 180,E1 -3284.531,E2 -3284.531} C_VEL
LIN {X 0,Y 552.137,Z 455.704,A -85,B 0,C 180,E1 -3287.584,E2 -3287.584} C_VEL
LIN {X 0,Y 552.135,Z 455.707,A -85,B 0,C 180,E1 -3290.472,E2 -3290.472} C_VEL
LIN {X 0,Y 552.105,Z 455.708,A -85,B 0,C 180,E1 -3293.318,E2 -3293.318} C_VEL
LIN {X 0,Y 552.107,Z 455.71,A -85,B 0,C 180,E1 -3295.937,E2 -3295.937} C_VEL
LIN {X 0,Y 552.127,Z 455.71,A -85,B 0,C 180,E1 -3298.54,E2 -3298.54} C_VEL
LIN {X 0,Y 552.102,Z 455.714,A -85,B 0,C 180,E1 -3301.443,E2 -3301.443} C_VEL
LIN {X 0,Y 552.164,Z 455.94,A -85,B 0,C 180,E1 -3302.278,E2 -3302.278} C_VEL
LIN {X 0,Y 554.187,Z 465.27,A -85,B 0,C 180,E1 -3303.446,E2 -3303.446} C_VEL
LIN {X 0,Y 553.911,Z 486.637,A -85,B 0,C 180,E1 -3305.865,E2 -3305.865} C_VEL
LIN {X 0,Y 553.618,Z 511.353,A -85,B 0,C 180,E1 -3308.593,E2 -3308.593} C_VEL
LIN {X 0,Y 553.227,Z 533.622,A -85,B 0,C 180,E1 -3311.097,E2 -3311.097} C_VEL
LIN {X 0,Y 552.768,Z 558.939,A -85,B 0,C 180,E1 -3313.945,E2 -3313.945} C_VEL
LIN {X 0,Y 552.644,Z 573.859,A -85,B 0,C 180,E1 -3315.594,E2 -3315.594} C_VEL
LIN {X 0,Y 553.454,Z 581.422,A -85,B 0,C 180,E1 -3315.733,E2 -3315.733} C_VEL
LIN {X 0,Y 553.152,Z 683.89,A -85,B 0,C 180,E1 -3317.082,E2 -3317.082} C_VEL
LIN {X 0,Y 553.004,Z 697.181,A -85,B 0,C 180,E1 -3317.405,E2 -3317.405} C_VEL
LIN {X 0,Y 552.857,Z 709.342,A -85,B 0,C 180,E1 -3317.845,E2 -3317.845} C_VEL
LIN {X 0,Y 552.692,Z 721.651,A -85,B 0,C 180,E1 -3318.448,E2 -3318.448} C_VEL
LIN {X 0,Y 552.482,Z 733.182,A -85,B 0,C 180,E1 -3319.184,E2 -3319.184} C_VEL
LIN {X 0,Y 552.3,Z 743.59,A -85,B 0,C 180,E1 -3320.015,E2 -3320.015} C_VEL
LIN {X 0,Y 552.127,Z 752.102,A -85,B 0,C 180,E1 -3320.843,E2 -3320.843} C_VEL
LIN {X 0,Y 552.013,Z 759.951,A -85,B 0,C 180,E1 -3321.764,E2 -3321.764} C_VEL
LIN {X 0,Y 551.891,Z 767.614,A -85,B 0,C 180,E1 -3322.867,E2 -3322.867} C_VEL
LIN {X 0,Y 551.868,Z 774.674,A -85,B 0,C 180,E1 -3324.151,E2 -3324.151} C_VEL
LIN {X 0,Y 551.725,Z 779.368,A -85,B 0,C 180,E1 -3325.249,E2 -3325.249} C_VEL
LIN {X 0,Y 551.751,Z 782.954,A -85,B 0,C 180,E1 -3326.347,E2 -3326.347} C_VEL
LIN {X 0,Y 551.724,Z 784.805,A -85,B 0,C 180,E1 -3327.078,E2 -3327.078} C_VEL
LIN {X 0,Y 551.645,Z 787.183,A -85,B 0,C 180,E1 -3328.539,E2 -3328.539} C_VEL
LIN {X 0,Y 551.64,Z 788,A -85,B 0,C 180,E1 -3329.999,E2 -3329.999} C_VEL
LIN {X 0,Y 551.645,Z 787.187,A -85,B 0,C 180,E1 -3331.459,E2 -3331.459} C_VEL
LIN {X 0,Y 551.723,Z 784.813,A -85,B 0,C 180,E1 -3332.919,E2 -3332.919} C_VEL
LIN {X 0,Y 551.764,Z 781.899,A -85,B 0,C 180,E1 -3334.016,E2 -3334.016} C_VEL
LIN {X 0,Y 551.723,Z 777.953,A -85,B 0,C 180,E1 -3335.114,E2 -3335.114} C_VEL
LIN {X 0,Y 551.813,Z 772.136,A -85,B 0,C 180,E1 -3336.351,E2 -3336.351} C_VEL
LIN {X 0,Y 551.925,Z 765.245,A -85,B 0,C 180,E1 -3337.498,E2 -3337.498} C_VEL
LIN {X 0,Y 552.081,Z 757.002,A -85,B 0,C 180,E1 -3338.601,E2 -3338.601} C_VEL
LIN {X 0,Y 552.222,Z 748.552,A -85,B 0,C 180,E1 -3339.522,E2 -3339.522} C_VEL
LIN {X 0,Y 552.384,Z 738.112,A -85,B 0,C 180,E1 -3340.444,E2 -3340.444} C_VEL
LIN {X 0,Y 552.619,Z 727.151,A -85,B 0,C 180,E1 -3341.222,E2 -3341.222} C_VEL
LIN {X 0,Y 552.781,Z 716.433,A -85,B 0,C 180,E1 -3341.829,E2 -3341.829} C_VEL
LIN {X 0,Y 552.897,Z 704.801,A -85,B 0,C 180,E1 -3342.338,E2 -3342.338} C_VEL
LIN {X 0,Y 553.049,Z 691.399,A -85,B 0,C 180,E1 -3342.754,E2 -3342.754} C_VEL
LIN {X 0,Y 553.191,Z 678.178,A -85,B 0,C 180,E1 -3343.008,E2 -3343.008} C_VEL
LIN {X 0,Y 553.376,Z 579.825,A -85,B 0,C 180,E1 -3344.29,E2 -3344.29} C_VEL
LIN {X 0,Y 552.647,Z 573.931,A -85,B 0,C 180,E1 -3344.404,E2 -3344.404} C_VEL
LIN {X 0,Y 553.02,Z 545.203,A -85,B 0,C 180,E1 -3347.611,E2 -3347.611} C_VEL
LIN {X 0,Y 553.564,Z 516.936,A -85,B 0,C 180,E1 -3350.822,E2 -3350.822} C_VEL
LIN {X 0,Y 553.947,Z 488.216,A -85,B 0,C 180,E1 -3354.01,E2 -3354.01} C_VEL
LIN {X 0,Y 554.222,Z 465.876,A -85,B 0,C 180,E1 -3356.55,E2 -3356.55} C_VEL
LIN {X 0,Y 552.358,Z 456.901,A -85,B 0,C 180,E1 -3357.671,E2 -3357.671} C_VEL
LIN {X 0,Y 552.129,Z 455.838,A -85,B 0,C 180,E1 -3357.838,E2 -3357.838} C_VEL
LIN {X 0,Y 552.088,Z 455.714,A -85,B 0,C 180,E1 -3360.608,E2 -3360.608} C_VEL
LIN {X 0,Y 552.101,Z 455.709,A -85,B 0,C 180,E1 -3363.185,E2 -3363.185} C_VEL
LIN {X 0,Y 552.062,Z 455.718,A -85,B 0,C 180,E1 -3365.844,E2 -3365.844} C_VEL
LIN {X 0,Y 552.109,Z 455.706,A -85,B 0,C 180,E1 -3369.059,E2 -3369.059} C_VEL
LIN {X 0,Y 552.07,Z 455.711,A -85,B 0,C 180,E1 -3371.448,E2 -3371.448} C_VEL
LIN {X 0,Y 552.066,Z 455.718,A -85,B 0,C 180,E1 -3374.438,E2 -3374.438} C_VEL
LIN {X 0,Y 552.098,Z 455.709,A -85,B 0,C 180,E1 -3377.586,E2 -3377.586} C_VEL
LIN {X 0,Y 552.116,Z 455.711,A -85,B 0,C 180,E1 -3380.471,E2 -3380.471} C_VEL
LIN {X 0,Y 552.087,Z 455.709,A -85,B 0,C 180,E1 -3383.317,E2 -3383.317} C_VEL
LIN {X 0,Y 552.114,Z 455.71,A -85,B 0,C 180,E1 -3385.938,E2 -3385.938} C_VEL
LIN {X 0,Y 552.108,Z 455.712,A -85,B 0,C 180,E1 -3388.54,E2 -3388.54} C_VEL
LIN {X 0,Y 552.091,Z 455.708,A -85,B 0,C 180,E1 -3391.441,E2 -3391.441} C_VEL
LIN {X 0,Y 552.1,Z 455.707,A -85,B 0,C 180,E1 -3393.542,E2 -3393.542} C_VEL
LIN {X 0,Y 552.081,Z 455.719,A -85,B 0,C 180,E1 -3396.424,E2 -3396.424} C_VEL
LIN {X 0,Y 552.105,Z 455.707,A -85,B 0,C 180,E1 -3399.119,E2 -3399.119} C_VEL
LIN {X 0,Y 552.079,Z 455.71,A -85,B 0,C 180,E1 -3401.443,E2 -3401.443} C_VEL
LIN {X 0,Y 552.096,Z 455.708,A -85,B 0,C 180,E1 -3403.736,E2 -3403.736} C_VEL
LIN {X 0,Y 552.109,Z 455.709,A -85,B 0,C 180,E1 -3406.003,E2 -3406.003} C_VEL
LIN {X 0,Y 552.167,Z 455.701,A -85,B 0,C 180,E1 -3408.993,E2 -3408.993} C_VEL
LIN {X 0,Y 552.139,Z 455.704,A -85,B 0,C 180,E1 -3411.951,E2 -3411.951} C_VEL
LIN {X 0,Y 552.211,Z 455.697,A -85,B 0,C 180,E1 -3414.889,E2 -3414.889} C_VEL
LIN {X 0,Y 552.202,Z 455.695,A -85,B 0,C 180,E1 -3417.812,E2 -3417.812} C_VEL
LIN {X 0,Y 552.236,Z 455.697,A -85,B 0,C 180,E1 -3420.729,E2 -3420.729} C_VEL
LIN {X 0,Y 552.198,Z 455.699,A -85,B 0,C 180,E1 -3422.918,E2 -3422.918} C_VEL
LIN {X 0,Y 552.18,Z 455.698,A -85,B 0,C 180,E1 -3425.844,E2 -3425.844} C_VEL
LIN {X 0,Y 552.157,Z 455.707,A -85,B 0,C 180,E1 -3428.785,E2 -3428.785} C_VEL
LIN {X 0,Y 552.151,Z 455.701,A -85,B 0,C 180,E1 -3431.75,E2 -3431.75} C_VEL
LIN {X 0,Y 552.122,Z 455.713,A -85,B 0,C 180,E1 -3434.748,E2 -3434.748} C_VEL
LIN {X 0,Y 552.098,Z 455.707,A -85,B 0,C 180,E1 -3437.789,E2 -3437.789} C_VEL
LIN {X 0,Y 552.12,Z 455.706,A -85,B 0,C 180,E1 -3440.101,E2 -3440.101} C_VEL
LIN {X 0,Y 552.083,Z 455.715,A -85,B 0,C 180,E1 -3442.451,E2 -3442.451} C_VEL
LIN {X 0,Y 552.141,Z 455.703,A -85,B 0,C 180,E1 -3445.351,E2 -3445.351} C_VEL
LIN {X 0,Y 552.113,Z 455.707,A -85,B 0,C 180,E1 -3448.098,E2 -3448.098} C_VEL
LIN {X 0,Y 552.093,Z 455.715,A -85,B 0,C 180,E1 -3450.631,E2 -3450.631} C_VEL
LIN {X 0,Y 552.116,Z 455.709,A -85,B 0,C 180,E1 -3453.185,E2 -3453.185} C_VEL
LIN {X 0,Y 552.111,Z 455.706,A -85,B 0,C 180,E1 -3453.811,E2 -3453.811} C_VEL
LIN {X 0,Y 551.477,Z 455.79,A -85,B 0,C 180,E1 -3454.42,E2 -3454.42} C_VEL
LIN {X 0,Y 548.65,Z 456.148,A -85,B 0,C 180,E1 -3455.408,E2 -3455.408} C_VEL
LIN {X 0,Y 546.224,Z 456.453,A -85,B 0,C 180,E1 -3456.203,E2 -3456.203} C_VEL
LIN {X 0,Y 545.153,Z 456.583,A -85,B 0,C 180,E1 -3456.817,E2 -3456.817} C_VEL
LIN {X 0,Y 545.051,Z 456.592,A -85,B 0,C 180,E1 -3457.025,E2 -3457.025} C_VEL
LIN {X 0,Y 545.063,Z 456.585,A -85,B 0,C 180,E1 -3460.143,E2 -3460.143} C_VEL
LIN {X 0,Y 545.075,Z 456.588,A -85,B 0,C 180,E1 -3463.107,E2 -3463.107} C_VEL
LIN {X 0,Y 545.055,Z 456.586,A -85,B 0,C 180,E1 -3466.225,E2 -3466.225} C_VEL
LIN {X 0,Y 545.113,Z 456.587,A -85,B 0,C 180,E1 -3468.89,E2 -3468.89} C_VEL
LIN {X 0,Y 545.045,Z 456.586,A -85,B 0,C 180,E1 -3471.764,E2 -3471.764} C_VEL
LIN {X 0,Y 545.045,Z 456.589,A -85,B 0,C 180,E1 -3474.534,E2 -3474.534} C_VEL
LIN {X 0,Y 545.074,Z 456.588,A -85,B 0,C 180,E1 -3477.214,E2 -3477.214} C_VEL
LIN {X 0,Y 545.059,Z 456.584,A -85,B 0,C 180,E1 -3479.812,E2 -3479.812} C_VEL
LIN {X 0,Y 545.087,Z 456.582,A -85,B 0,C 180,E1 -3482.346,E2 -3482.346} C_VEL
LIN {X 0,Y 545.111,Z 456.584,A -85,B 0,C 180,E1 -3484.822,E2 -3484.822} C_VEL
LIN {X 0,Y 545.039,Z 456.593,A -85,B 0,C 180,E1 -3487.244,E2 -3487.244} C_VEL
LIN {X 0,Y 545.115,Z 456.578,A -85,B 0,C 180,E1 -3490.416,E2 -3490.416} C_VEL
LIN {X 0,Y 545.072,Z 456.586,A -85,B 0,C 180,E1 -3493.523,E2 -3493.523} C_VEL
LIN {X 0,Y 545.092,Z 456.581,A -85,B 0,C 180,E1 -3495.821,E2 -3495.821} C_VEL
LIN {X 0,Y 545.115,Z 456.583,A -85,B 0,C 180,E1 -3498.851,E2 -3498.851} C_VEL
LIN {X 0,Y 545.128,Z 456.578,A -85,B 0,C 180,E1 -3501.848,E2 -3501.848} C_VEL
LIN {X 0,Y 545.206,Z 456.572,A -85,B 0,C 180,E1 -3504.824,E2 -3504.824} C_VEL
LIN {X 0,Y 545.197,Z 456.573,A -85,B 0,C 180,E1 -3507.785,E2 -3507.785} C_VEL
LIN {X 0,Y 545.221,Z 456.697,A -85,B 0,C 180,E1 -3509.724,E2 -3509.724} C_VEL
LIN {X 0,Y 545.341,Z 457.442,A -85,B 0,C 180,E1 -3509.84,E2 -3509.84} C_VEL
LIN {X 0,Y 546.579,Z 461.683,A -85,B 0,C 180,E1 -3509.955,E2 -3509.955} C_VEL
LIN {X 0,Y 546.351,Z 536.947,A -85,B 0,C 180,E1 -3510.969,E2 -3510.969} C_VEL
LIN {X 0,Y 546.219,Z 549.989,A -85,B 0,C 180,E1 -3511.291,E2 -3511.291} C_VEL
LIN {X 0,Y 546.076,Z 562.473,A -85,B 0,C 180,E1 -3511.753,E2 -3511.753} C_VEL
LIN {X 0,Y 545.942,Z 573.578,A -85,B 0,C 180,E1 -3512.307,E2 -3512.307} C_VEL
LIN {X 0,Y 545.716,Z 585.055,A -85,B 0,C 180,E1 -3513.046,E2 -3513.046} C_VEL
LIN {X 0,Y 545.498,Z 595.357,A -85,B 0,C 180,E1 -3513.88,E2 -3513.88} C_VEL
LIN {X 0,Y 545.31,Z 604.655,A -85,B 0,C 180,E1 -3514.807,E2 -3514.807} C_VEL
LIN {X 0,Y 545.117,Z 613.613,A -85,B 0,C 180,E1 -3515.921,E2 -3515.921} C_VEL
LIN {X 0,Y 545.043,Z 620.813,A -85,B 0,C 180,E1 -3517.037,E2 -3517.037} C_VEL
LIN {X 0,Y 544.891,Z 626.63,A -85,B 0,C 180,E1 -3518.158,E2 -3518.158} C_VEL
LIN {X 0,Y 544.792,Z 631.22,A -85,B 0,C 180,E1 -3519.281,E2 -3519.281} C_VEL
LIN {X 0,Y 544.743,Z 634.716,A -85,B 0,C 180,E1 -3520.407,E2 -3520.407} C_VEL
LIN {X 0,Y 544.704,Z 636.783,A -85,B 0,C 180,E1 -3521.311,E2 -3521.311} C_VEL
LIN {X 0,Y 544.679,Z 638.772,A -85,B 0,C 180,E1 -3522.672,E2 -3522.672} C_VEL
LIN {X 0,Y 544.631,Z 639.333,A -85,B 0,C 180,E1 -3523.432,E2 -3523.432} C_VEL
LIN {X 0,Y 544.634,Z 639.363,A -85,B 0,C 180,E1 -3524.579,E2 -3524.579} C_VEL
LIN {X 0,Y 544.633,Z 638.467,A -85,B 0,C 180,E1 -3525.724,E2 -3525.724} C_VEL
LIN {X 0,Y 544.654,Z 637.35,A -85,B 0,C 180,E1 -3526.493,E2 -3526.493} C_VEL
LIN {X 0,Y 544.719,Z 635.676,A -85,B 0,C 180,E1 -3527.303,E2 -3527.303} C_VEL
LIN {X 0,Y 544.749,Z 632.544,A -85,B 0,C 180,E1 -3528.427,E2 -3528.427} C_VEL
LIN {X 0,Y 544.863,Z 627.807,A -85,B 0,C 180,E1 -3529.679,E2 -3529.679} C_VEL
LIN {X 0,Y 544.955,Z 622.46,A -85,B 0,C 180,E1 -3530.773,E2 -3530.773} C_VEL
LIN {X 0,Y 545.137,Z 615.185,A -85,B 0,C 180,E1 -3531.956,E2 -3531.956} C_VEL
LIN {X 0,Y 545.265,Z 607.614,A -85,B 0,C 180,E1 -3532.949,E2 -3532.949} C_VEL
LIN {X 0,Y 545.464,Z 598.534,A -85,B 0,C 180,E1 -3533.921,E2 -3533.921} C_VEL
LIN {X 0,Y 545.591,Z 589.073,A -85,B 0,C 180,E1 -3534.75,E2 -3534.75} C_VEL
LIN {X 0,Y 545.868,Z 578.303,A -85,B 0,C 180,E1 -3535.508,E2 -3535.508} C_VEL
LIN {X 0,Y 546.051,Z 566.484,A -85,B 0,C 180,E1 -3536.157,E2 -3536.157} C_VEL
LIN {X 0,Y 546.146,Z 554.197,A -85,B 0,C 180,E1 -3536.667,E2 -3536.667} C_VEL
LIN {X 0,Y 546.298,Z 541.391,A -85,B 0,C 180,E1 -3537.033,E2 -3537.033} C_VEL
LIN {X 0,Y 546.329,Z 524.778,A -85,B 0,C 180,E1 -3537.303,E2 -3537.303} C_VEL
LIN {X 0,Y 546.518,Z 461.162,A -85,B 0,C 180,E1 -3538.146,E2 -3538.146} C_VEL
LIN {X 0,Y 545.255,Z 457.427,A -85,B 0,C 180,E1 -3538.258,E2 -3538.258} C_VEL
LIN {X 0,Y 545.093,Z 456.68,A -85,B 0,C 180,E1 -3538.389,E2 -3538.389} C_VEL
LIN {X 0,Y 545.07,Z 456.592,A -85,B 0,C 180,E1 -3541.049,E2 -3541.049} C_VEL
LIN {X 0,Y 545.053,Z 456.588,A -85,B 0,C 180,E1 -3543.674,E2 -3543.674} C_VEL
LIN {X 0,Y 545.074,Z 456.59,A -85,B 0,C 180,E1 -3546.927,E2 -3546.927} C_VEL
LIN {X 0,Y 545.069,Z 456.584,A -85,B 0,C 180,E1 -3550.144,E2 -3550.144} C_VEL
LIN {X 0,Y 545.083,Z 456.588,A -85,B 0,C 180,E1 -3553.107,E2 -3553.107} C_VEL
LIN {X 0,Y 545.053,Z 456.588,A -85,B 0,C 180,E1 -3556.227,E2 -3556.227} C_VEL
LIN {X 0,Y 545.085,Z 456.591,A -85,B 0,C 180,E1 -3558.886,E2 -3558.886} C_VEL
LIN {X 0,Y 545.054,Z 456.589,A -85,B 0,C 180,E1 -3561.763,E2 -3561.763} C_VEL
LIN {X 0,Y 545.115,Z 456.822,A -85,B 0,C 180,E1 -3563.452,E2 -3563.452} C_VEL
LIN {X 0,Y 546.165,Z 462.728,A -85,B 0,C 180,E1 -3564.407,E2 -3564.407} C_VEL
LIN {X 0,Y 545.98,Z 477.395,A -85,B 0,C 180,E1 -3566.639,E2 -3566.639} C_VEL
LIN {X 0,Y 545.712,Z 494.149,A -85,B 0,C 180,E1 -3569.181,E2 -3569.181} C_VEL
LIN {X 0,Y 545.392,Z 512.295,A -85,B 0,C 180,E1 -3571.944,E2 -3571.944} C_VEL
LIN {X 0,Y 545.447,Z 516.536,A -85,B 0,C 180,E1 -3572.48,E2 -3572.48} C_VEL
LIN {X 0,Y 546.583,Z 524.532,A -85,B 0,C 180,E1 -3572.636,E2 -3572.636} C_VEL
LIN {X 0,Y 546.213,Z 623.25,A -85,B 0,C 180,E1 -3573.955,E2 -3573.955} C_VEL
LIN {X 0,Y 546.067,Z 636.106,A -85,B 0,C 180,E1 -3574.253,E2 -3574.253} C_VEL
LIN {X 0,Y 545.856,Z 648.485,A -85,B 0,C 180,E1 -3574.697,E2 -3574.697} C_VEL
LIN {X 0,Y 545.756,Z 658.149,A -85,B 0,C 180,E1 -3575.158,E2 -3575.158} C_VEL
LIN {X 0,Y 545.564,Z 667.962,A -85,B 0,C 180,E1 -3575.734,E2 -3575.734} C_VEL
LIN {X 0,Y 545.375,Z 677.98,A -85,B 0,C 180,E1 -3576.454,E2 -3576.454} C_VEL
LIN {X 0,Y 545.179,Z 687.027,A -85,B 0,C 180,E1 -3577.249,E2 -3577.249} C_VEL
LIN {X 0,Y 545.005,Z 695.832,A -85,B 0,C 180,E1 -3578.198,E2 -3578.198} C_VEL
LIN {X 0,Y 544.89,Z 702.299,A -85,B 0,C 180,E1 -3579.028,E2 -3579.028} C_VEL
LIN {X 0,Y 544.803,Z 708.966,A -85,B 0,C 180,E1 -3580.05,E2 -3580.05} C_VEL
LIN {X 0,Y 544.733,Z 714.992,A -85,B 0,C 180,E1 -3581.184,E2 -3581.184} C_VEL
LIN {X 0,Y 544.655,Z 719.905,A -85,B 0,C 180,E1 -3582.387,E2 -3582.387} C_VEL
LIN {X 0,Y 544.614,Z 723.359,A -85,B 0,C 180,E1 -3583.507,E2 -3583.507} C_VEL
LIN {X 0,Y 544.553,Z 725.179,A -85,B 0,C 180,E1 -3584.275,E2 -3584.275} C_VEL
LIN {X 0,Y 544.562,Z 727.028,A -85,B 0,C 180,E1 -3585.454,E2 -3585.454} C_VEL
LIN {X 0,Y 544.557,Z 727.862,A -85,B 0,C 180,E1 -3586.567,E2 -3586.567} C_VEL
LIN {X 0,Y 544.57,Z 727.933,A -85,B 0,C 180,E1 -3587.327,E2 -3587.327} C_VEL
LIN {X 0,Y 544.569,Z 727.607,A -85,B 0,C 180,E1 -3588.084,E2 -3588.084} C_VEL
LIN {X 0,Y 544.612,Z 726.803,A -85,B 0,C 180,E1 -3588.839,E2 -3588.839} C_VEL
LIN {X 0,Y 544.606,Z 723.979,A -85,B 0,C 180,E1 -3590.343,E2 -3590.343} C_VEL
LIN {X 0,Y 544.671,Z 720.702,A -85,B 0,C 180,E1 -3591.467,E2 -3591.467} C_VEL
LIN {X 0,Y 544.704,Z 716.395,A -85,B 0,C 180,E1 -3592.587,E2 -3592.587} C_VEL
LIN {X 0,Y 544.768,Z 710.042,A -85,B 0,C 180,E1 -3593.862,E2 -3593.862} C_VEL
LIN {X 0,Y 544.859,Z 702.706,A -85,B 0,C 180,E1 -3595.005,E2 -3595.005} C_VEL
LIN {X 0,Y 544.987,Z 695.497,A -85,B 0,C 180,E1 -3595.933,E2 -3595.933} C_VEL
LIN {X 0,Y 545.215,Z 685.85,A -85,B 0,C 180,E1 -3596.952,E2 -3596.952} C_VEL
LIN {X 0,Y 545.409,Z 676.019,A -85,B 0,C 180,E1 -3597.785,E2 -3597.785} C_VEL
LIN {X 0,Y 545.595,Z 665.373,A -85,B 0,C 180,E1 -3598.524,E2 -3598.524} C_VEL
LIN {X 0,Y 545.753,Z 653.505,A -85,B 0,C 180,E1 -3599.17,E2 -3599.17} C_VEL
LIN {X 0,Y 546.035,Z 642.185,A -85,B 0,C 180,E1 -3599.632,E2 -3599.632} C_VEL
LIN {X 0,Y 546.125,Z 631.606,A -85,B 0,C 180,E1 -3599.954,E2 -3599.954} C_VEL
LIN {X 0,Y 546.239,Z 619.05,A -85,B 0,C 180,E1 -3600.208,E2 -3600.208} C_VEL
LIN {X 0,Y 546.452,Z 523.301,A -85,B 0,C 180,E1 -3601.474,E2 -3601.474} C_VEL
LIN {X 0,Y 545.43,Z 516.497,A -85,B 0,C 180,E1 -3601.615,E2 -3601.615} C_VEL
LIN {X 0,Y 545.417,Z 513.09,A -85,B 0,C 180,E1 -3602.031,E2 -3602.031} C_VEL
LIN {X 0,Y 545.66,Z 495.005,A -85,B 0,C 180,E1 -3604.803,E2 -3604.803} C_VEL
LIN {X 0,Y 545.946,Z 480.211,A -85,B 0,C 180,E1 -3607.025,E2 -3607.025} C_VEL
LIN {X 0,Y 546.209,Z 463.077,A -85,B 0,C 180,E1 -3609.629,E2 -3609.629} C_VEL
LIN {X 0,Y 545.137,Z 456.669,A -85,B 0,C 180,E1 -3610.633,E2 -3610.633} C_VEL
LIN {X 0,Y 545.054,Z 456.594,A -85,B 0,C 180,E1 -3613.421,E2 -3613.421} C_VEL
LIN {X 0,Y 545.049,Z 456.59,A -85,B 0,C 180,E1 -3615.711,E2 -3615.711} C_VEL
LIN {X 0,Y 545.062,Z 456.586,A -85,B 0,C 180,E1 -3618.027,E2 -3618.027} C_VEL
LIN {X 0,Y 545.097,Z 456.583,A -85,B 0,C 180,E1 -3620.372,E2 -3620.372} C_VEL
LIN {X 0,Y 545.081,Z 456.585,A -85,B 0,C 180,E1 -3623.56,E2 -3623.56} C_VEL
LIN {X 0,Y 545.076,Z 456.584,A -85,B 0,C 180,E1 -3626.001,E2 -3626.001} C_VEL
LIN {X 0,Y 545.095,Z 456.589,A -85,B 0,C 180,E1 -3628.747,E2 -3628.747} C_VEL
LIN {X 0,Y 545.063,Z 456.585,A -85,B 0,C 180,E1 -3631.915,E2 -3631.915} C_VEL
LIN {X 0,Y 545.071,Z 456.591,A -85,B 0,C 180,E1 -3634.564,E2 -3634.564} C_VEL
LIN {X 0,Y 545.044,Z 456.588,A -85,B 0,C 180,E1 -3637.304,E2 -3637.304} C_VEL
LIN {X 0,Y 545.074,Z 456.587,A -85,B 0,C 180,E1 -3640.142,E2 -3640.142} C_VEL
LIN {X 0,Y 545.086,Z 456.584,A -85,B 0,C 180,E1 -3643.106,E2 -3643.106} C_VEL
LIN {X 0,Y 545.057,Z 456.593,A -85,B 0,C 180,E1 -3646.226,E2 -3646.226} C_VEL
LIN {X 0,Y 545.089,Z 456.584,A -85,B 0,C 180,E1 -3648.885,E2 -3648.885} C_VEL
LIN {X 0,Y 545.054,Z 456.585,A -85,B 0,C 180,E1 -3651.864,E2 -3651.864} C_VEL
LIN {X 0,Y 545.033,Z 456.591,A -85,B 0,C 180,E1 -3654.53,E2 -3654.53} C_VEL
LIN {X 0,Y 545.071,Z 456.586,A -85,B 0,C 180,E1 -3657.211,E2 -3657.211} C_VEL
LIN {X 0,Y 545.068,Z 456.591,A -85,B 0,C 180,E1 -3659.81,E2 -3659.81} C_VEL
LIN {X 0,Y 545.091,Z 456.78,A -85,B 0,C 180,E1 -3662.082,E2 -3662.082} C_VEL
LIN {X 0,Y 547.201,Z 466.198,A -85,B 0,C 180,E1 -3663.286,E2 -3663.286} C_VEL
LIN {X 0,Y 547.042,Z 480.284,A -85,B 0,C 180,E1 -3664.914,E2 -3664.914} C_VEL
LIN {X 0,Y 546.733,Z 504.23,A -85,B 0,C 180,E1 -3667.619,E2 -3667.619} C_VEL
LIN {X 0,Y 546.376,Z 527.288,A -85,B 0,C 180,E1 -3670.177,E2 -3670.177} C_VEL
LIN {X 0,Y 546.062,Z 548.762,A -85,B 0,C 180,E1 -3672.582,E2 -3672.582} C_VEL
LIN {X 0,Y 545.671,Z 573.902,A -85,B 0,C 180,E1 -3675.408,E2 -3675.408} C_VEL
LIN {X 0,Y 546.573,Z 581.547,A -85,B 0,C 180,E1 -3675.551,E2 -3675.551} C_VEL
LIN {X 0,Y 546.241,Z 683.89,A -85,B 0,C 180,E1 -3676.916,E2 -3676.916} C_VEL
LIN {X 0,Y 546.085,Z 696.418,A -85,B 0,C 180,E1 -3677.219,E2 -3677.219} C_VEL
LIN {X 0,Y 545.926,Z 709.342,A -85,B 0,C 180,E1 -3677.688,E2 -3677.688} C_VEL
LIN {X 0,Y 545.734,Z 721.65,A -85,B 0,C 180,E1 -3678.299,E2 -3678.299} C_VEL
LIN {X 0,Y 545.495,Z 733.18,A -85,B 0,C 180,E1 -3679.044,E2 -3679.044} C_VEL
LIN {X 0,Y 545.263,Z 743.591,A -85,B 0,C 180,E1 -3679.884,E2 -3679.884} C_VEL
LIN {X 0,Y 545.086,Z 752.102,A -85,B 0,C 180,E1 -3680.724,E2 -3680.724} C_VEL
LIN {X 0,Y 544.977,Z 759.951,A -85,B 0,C 180,E1 -3681.657,E2 -3681.657} C_VEL
LIN {X 0,Y 544.825,Z 767.614,A -85,B 0,C 180,E1 -3682.774,E2 -3682.774} C_VEL
LIN {X 0,Y 544.777,Z 774.674,A -85,B 0,C 180,E1 -3684.075,E2 -3684.075} C_VEL
LIN {X 0,Y 544.629,Z 779.368,A -85,B 0,C 180,E1 -3685.187,E2 -3685.187} C_VEL
LIN {X 0,Y 544.669,Z 782.955,A -85,B 0,C 180,E1 -3686.3,E2 -3686.3} C_VEL
LIN {X 0,Y 544.651,Z 784.805,A -85,B 0,C 180,E1 -3687.04,E2 -3687.04} C_VEL
LIN {X 0,Y 544.546,Z 787.182,A -85,B 0,C 180,E1 -3688.52,E2 -3688.52} C_VEL
LIN {X 0,Y 544.541,Z 788,A -85,B 0,C 180,E1 -3689.999,E2 -3689.999} C_VEL
LIN {X 0,Y 544.546,Z 787.186,A -85,B 0,C 180,E1 -3691.478,E2 -3691.478} C_VEL
LIN {X 0,Y 544.65,Z 784.813,A -85,B 0,C 180,E1 -3692.957,E2 -3692.957} C_VEL
LIN {X 0,Y 544.684,Z 781.899,A -85,B 0,C 180,E1 -3694.068,E2 -3694.068} C_VEL
LIN {X 0,Y 544.653,Z 777.953,A -85,B 0,C 180,E1 -3695.181,E2 -3695.181} C_VEL
LIN {X 0,Y 544.728,Z 772.656,A -85,B 0,C 180,E1 -3696.337,E2 -3696.337} C_VEL
LIN {X 0,Y 544.858,Z 765.245,A -85,B 0,C 180,E1 -3697.596,E2 -3697.596} C_VEL
LIN {X 0,Y 545.028,Z 757.002,A -85,B 0,C 180,E1 -3698.713,E2 -3698.713} C_VEL
LIN {X 0,Y 545.202,Z 748.553,A -85,B 0,C 180,E1 -3699.646,E2 -3699.646} C_VEL
LIN {X 0,Y 545.38,Z 738.111,A -85,B 0,C 180,E1 -3700.58,E2 -3700.58} C_VEL
LIN {X 0,Y 545.634,Z 726.374,A -85,B 0,C 180,E1 -3701.419,E2 -3701.419} C_VEL
LIN {X 0,Y 545.845,Z 714.517,A -85,B 0,C 180,E1 -3702.076,E2 -3702.076} C_VEL
LIN {X 0,Y 546.016,Z 702.204,A -85,B 0,C 180,E1 -3702.591,E2 -3702.591} C_VEL
LIN {X 0,Y 546.137,Z 689.569,A -85,B 0,C 180,E1 -3702.966,E2 -3702.966} C_VEL
LIN {X 0,Y 546.284,Z 676.414,A -85,B 0,C 180,E1 -3703.199,E2 -3703.199} C_VEL
LIN {X 0,Y 546.431,Z 579.865,A -85,B 0,C 180,E1 -3704.475,E2 -3704.475} C_VEL
LIN {X 0,Y 545.661,Z 573.95,A -85,B 0,C 180,E1 -3704.591,E2 -3704.591} C_VEL
LIN {X 0,Y 546.097,Z 545.917,A -85,B 0,C 180,E1 -3707.759,E2 -3707.759} C_VEL
LIN {X 0,Y 546.54,Z 519.577,A -85,B 0,C 180,E1 -3710.708,E2 -3710.708} C_VEL
LIN {X 0,Y 546.955,Z 491.62,A -85,B 0,C 180,E1 -3713.847,E2 -3713.847} C_VEL
LIN {X 0,Y 547.33,Z 468.613,A -85,B 0,C 180,E1 -3716.499,E2 -3716.499} C_VEL
LIN {X 0,Y 547.079,Z 465.389,A -85,B 0,C 180,E1 -3716.887,E2 -3716.887} C_VEL
LIN {X 0,Y 545.099,Z 456.735,A -85,B 0,C 180,E1 -3718.019,E2 -3718.019} C_VEL
LIN {X 0,Y 545.057,Z 456.588,A -85,B 0,C 180,E1 -3721.047,E2 -3721.047} C_VEL
LIN {X 0,Y 545.051,Z 456.59,A -85,B 0,C 180,E1 -3723.671,E2 -3723.671} C_VEL
LIN {X 0,Y 545.029,Z 456.588,A -85,B 0,C 180,E1 -3726.92,E2 -3726.92} C_VEL
LIN {X 0,Y 545.064,Z 456.584,A -85,B 0,C 180,E1 -3729.318,E2 -3729.318} C_VEL
LIN {X 0,Y 545.045,Z 456.594,A -85,B 0,C 180,E1 -3732.104,E2 -3732.104} C_VEL
LIN {X 0,Y 545.02,Z 456.589,A -85,B 0,C 180,E1 -3735.169,E2 -3735.169} C_VEL
LIN {X 0,Y 545.051,Z 456.59,A -85,B 0,C 180,E1 -3737.894,E2 -3737.894} C_VEL
LIN {X 0,Y 545.066,Z 456.585,A -85,B 0,C 180,E1 -3740.817,E2 -3740.817} C_VEL
LIN {X 0,Y 545.023,Z 456.59,A -85,B 0,C 180,E1 -3743.618,E2 -3743.618} C_VEL
LIN {X 0,Y 545.053,Z 456.595,A -85,B 0,C 180,E1 -3746.327,E2 -3746.327} C_VEL
LIN {X 0,Y 545.053,Z 456.586,A -85,B 0,C 180,E1 -3748.951,E2 -3748.951} C_VEL
LIN {X 0,Y 545.07,Z 456.583,A -85,B 0,C 180,E1 -3751.506,E2 -3751.506} C_VEL
LIN {X 0,Y 545.056,Z 456.592,A -85,B 0,C 180,E1 -3754.496,E2 -3754.496} C_VEL
LIN {X 0,Y 545.019,Z 456.589,A -85,B 0,C 180,E1 -3757.241,E2 -3757.241} C_VEL
LIN {X 0,Y 545.104,Z 456.589,A -85,B 0,C 180,E1 -3760.414,E2 -3760.414} C_VEL
LIN {X 0,Y 545.048,Z 456.586,A -85,B 0,C 180,E1 -3763.52,E2 -3763.52} C_VEL
LIN {X 0,Y 545.07,Z 456.584,A -85,B 0,C 180,E1 -3765.819,E2 -3765.819} C_VEL
LIN {X 0,Y 545.121,Z 456.58,A -85,B 0,C 180,E1 -3768.849,E2 -3768.849} C_VEL
LIN {X 0,Y 545.109,Z 456.579,A -85,B 0,C 180,E1 -3771.846,E2 -3771.846} C_VEL
LIN {X 0,Y 545.186,Z 456.573,A -85,B 0,C 180,E1 -3774.822,E2 -3774.822} C_VEL
LIN {X 0,Y 545.174,Z 456.57,A -85,B 0,C 180,E1 -3777.783,E2 -3777.783} C_VEL
LIN {X 0,Y 545.205,Z 456.573,A -85,B 0,C 180,E1 -3780.738,E2 -3780.738} C_VEL
LIN {X 0,Y 545.163,Z 456.575,A -85,B 0,C 180,E1 -3782.956,E2 -3782.956} C_VEL
LIN {X 0,Y 545.152,Z 456.574,A -85,B 0,C 180,E1 -3785.919,E2 -3785.919} C_VEL
LIN {X 0,Y 545.114,Z 456.583,A -85,B 0,C 180,E1 -3788.9,E2 -3788.9} C_VEL
LIN {X 0,Y 545.122,Z 456.577,A -85,B 0,C 180,E1 -3791.904,E2 -3791.904} C_VEL
LIN {X 0,Y 545.072,Z 456.588,A -85,B 0,C 180,E1 -3794.944,E2 -3794.944} C_VEL
LIN {X 0,Y 545.066,Z 456.584,A -85,B 0,C 180,E1 -3798.026,E2 -3798.026} C_VEL
LIN {X 0,Y 545.085,Z 456.586,A -85,B 0,C 180,E1 -3800.372,E2 -3800.372} C_VEL
LIN {X 0,Y 545.077,Z 456.582,A -85,B 0,C 180,E1 -3803.559,E2 -3803.559} C_VEL
LIN {X 0,Y 545.067,Z 456.584,A -85,B 0,C 180,E1 -3806.001,E2 -3806.001} C_VEL
LIN {X 0,Y 545.078,Z 456.592,A -85,B 0,C 180,E1 -3808.749,E2 -3808.749} C_VEL
LIN {X 0,Y 545.065,Z 456.583,A -85,B 0,C 180,E1 -3811.683,E2 -3811.683} C_VEL
LIN {X 0,Y 545.072,Z 456.589,A -85,B 0,C 180,E1 -3814.563,E2 -3814.563} C_VEL
LIN {X 0,Y 545.051,Z 456.592,A -85,B 0,C 180,E1 -3817.025,E2 -3817.025} C_VEL
LIN {X 0,Y 544.344,Z 456.676,A -85,B 0,C 180,E1 -3817.641,E2 -3817.641} C_VEL
LIN {X 0,Y 541.481,Z 457.037,A -85,B 0,C 180,E1 -3818.642,E2 -3818.642} C_VEL
LIN {X 0,Y 539.095,Z 457.329,A -85,B 0,C 180,E1 -3819.448,E2 -3819.448} C_VEL
LIN {X 0,Y 538.086,Z 457.453,A -85,B 0,C 180,E1 -3820.07,E2 -3820.07} C_VEL
LIN {X 0,Y 538.01,Z 457.464,A -85,B 0,C 180,E1 -3820.28,E2 -3820.28} C_VEL
LIN {X 0,Y 538.022,Z 457.469,A -85,B 0,C 180,E1 -3822.989,E2 -3822.989} C_VEL
LIN {X 0,Y 538.019,Z 457.461,A -85,B 0,C 180,E1 -3825.926,E2 -3825.926} C_VEL
LIN {X 0,Y 538.07,Z 457.459,A -85,B 0,C 180,E1 -3829.25,E2 -3829.25} C_VEL
LIN {X 0,Y 537.985,Z 457.466,A -85,B 0,C 180,E1 -3832.124,E2 -3832.124} C_VEL
LIN {X 0,Y 538.004,Z 457.473,A -85,B 0,C 180,E1 -3834.918,E2 -3834.918} C_VEL
LIN {X 0,Y 538.024,Z 457.462,A -85,B 0,C 180,E1 -3837.619,E2 -3837.619} C_VEL
LIN {X 0,Y 538.011,Z 457.463,A -85,B 0,C 180,E1 -3840.24,E2 -3840.24} C_VEL
LIN {X 0,Y 538.06,Z 457.462,A -85,B 0,C 180,E1 -3842.798,E2 -3842.798} C_VEL
LIN {X 0,Y 538.043,Z 457.464,A -85,B 0,C 180,E1 -3845.294,E2 -3845.294} C_VEL
LIN {X 0,Y 538.009,Z 457.462,A -85,B 0,C 180,E1 -3848.043,E2 -3848.043} C_VEL
LIN {X 0,Y 538.034,Z 457.467,A -85,B 0,C 180,E1 -3850.941,E2 -3850.941} C_VEL
LIN {X 0,Y 538.023,Z 457.467,A -85,B 0,C 180,E1 -3853.3,E2 -3853.3} C_VEL
LIN {X 0,Y 538.06,Z 457.458,A -85,B 0,C 180,E1 -3855.632,E2 -3855.632} C_VEL
LIN {X 0,Y 538.074,Z 457.458,A -85,B 0,C 180,E1 -3858.703,E2 -3858.703} C_VEL
LIN {X 0,Y 538.085,Z 457.456,A -85,B 0,C 180,E1 -3861.741,E2 -3861.741} C_VEL
LIN {X 0,Y 538.163,Z 457.449,A -85,B 0,C 180,E1 -3864.756,E2 -3864.756} C_VEL
LIN {X 0,Y 538.168,Z 457.45,A -85,B 0,C 180,E1 -3867.756,E2 -3867.756} C_VEL
LIN {X 0,Y 538.177,Z 457.609,A -85,B 0,C 180,E1 -3869.541,E2 -3869.541} C_VEL
LIN {X 0,Y 538.421,Z 458.737,A -85,B 0,C 180,E1 -3869.673,E2 -3869.673} C_VEL
LIN {X 0,Y 539.719,Z 462.571,A -85,B 0,C 180,E1 -3869.772,E2 -3869.772} C_VEL
LIN {X 0,Y 539.478,Z 537.641,A -85,B 0,C 180,E1 -3870.794,E2 -3870.794} C_VEL
LIN {X 0,Y 539.36,Z 550.754,A -85,B 0,C 180,E1 -3871.121,E2 -3871.121} C_VEL
LIN {X 0,Y 539.207,Z 563.286,A -85,B 0,C 180,E1 -3871.588,E2 -3871.588} C_VEL
LIN {X 0,Y 539.075,Z 574.422,A -85,B 0,C 180,E1 -3872.149,E2 -3872.149} C_VEL
LIN {X 0,Y 538.819,Z 585.935,A -85,B 0,C 180,E1 -3872.898,E2 -3872.898} C_VEL
LIN {X 0,Y 538.591,Z 596.248,A -85,B 0,C 180,E1 -3873.742,E2 -3873.742} C_VEL
LIN {X 0,Y 538.379,Z 605.562,A -85,B 0,C 180,E1 -3874.681,E2 -3874.681} C_VEL
LIN {X 0,Y 538.165,Z 614.537,A -85,B 0,C 180,E1 -3875.81,E2 -3875.81} C_VEL
LIN {X 0,Y 538.063,Z 621.724,A -85,B 0,C 180,E1 -3876.936,E2 -3876.936} C_VEL
LIN {X 0,Y 537.878,Z 628.427,A -85,B 0,C 180,E1 -3878.265,E2 -3878.265} C_VEL
LIN {X 0,Y 537.775,Z 632.826,A -85,B 0,C 180,E1 -3879.403,E2 -3879.403} C_VEL
LIN {X 0,Y 537.728,Z 636.161,A -85,B 0,C 180,E1 -3880.544,E2 -3880.544} C_VEL
LIN {X 0,Y 537.693,Z 637.982,A -85,B 0,C 180,E1 -3881.394,E2 -3881.394} C_VEL
LIN {X 0,Y 537.637,Z 639.944,A -85,B 0,C 180,E1 -3882.841,E2 -3882.841} C_VEL
LIN {X 0,Y 537.6,Z 640.364,A -85,B 0,C 180,E1 -3883.611,E2 -3883.611} C_VEL
LIN {X 0,Y 537.625,Z 640.31,A -85,B 0,C 180,E1 -3884.682,E2 -3884.682} C_VEL
LIN {X 0,Y 537.622,Z 639.224,A -85,B 0,C 180,E1 -3885.935,E2 -3885.935} C_VEL
LIN {X 0,Y 537.725,Z 636.471,A -85,B 0,C 180,E1 -3887.428,E2 -3887.428} C_VEL
LIN {X 0,Y 537.785,Z 632.917,A -85,B 0,C 180,E1 -3888.675,E2 -3888.675} C_VEL
LIN {X 0,Y 537.89,Z 628.343,A -85,B 0,C 180,E1 -3889.861,E2 -3889.861} C_VEL
LIN {X 0,Y 538.036,Z 622.393,A -85,B 0,C 180,E1 -3891.053,E2 -3891.053} C_VEL
LIN {X 0,Y 538.18,Z 614.809,A -85,B 0,C 180,E1 -3892.255,E2 -3892.255} C_VEL
LIN {X 0,Y 538.351,Z 606.951,A -85,B 0,C 180,E1 -3893.261,E2 -3893.261} C_VEL
LIN {X 0,Y 538.599,Z 597.089,A -85,B 0,C 180,E1 -3894.283,E2 -3894.283} C_VEL
LIN {X 0,Y 538.821,Z 586.155,A -85,B 0,C 180,E1 -3895.186,E2 -3895.186} C_VEL
LIN {X 0,Y 539.079,Z 575.247,A -85,B 0,C 180,E1 -3895.901,E2 -3895.901} C_VEL
LIN {X 0,Y 539.213,Z 563.149,A -85,B 0,C 180,E1 -3896.515,E2 -3896.515} C_VEL
LIN {X 0,Y 539.378,Z 550.688,A -85,B 0,C 180,E1 -3896.976,E2 -3896.976} C_VEL
LIN {X 0,Y 539.477,Z 538.109,A -85,B 0,C 180,E1 -3897.29,E2 -3897.29} C_VEL
LIN {X 0,Y 539.646,Z 462.576,A -85,B 0,C 180,E1 -3898.323,E2 -3898.323} C_VEL
LIN {X 0,Y 538.215,Z 458.368,A -85,B 0,C 180,E1 -3898.445,E2 -3898.445} C_VEL
LIN {X 0,Y 538.067,Z 457.557,A -85,B 0,C 180,E1 -3898.581,E2 -3898.581} C_VEL
LIN {X 0,Y 538.012,Z 457.466,A -85,B 0,C 180,E1 -3901.502,E2 -3901.502} C_VEL
LIN {X 0,Y 538.014,Z 457.465,A -85,B 0,C 180,E1 -3904.175,E2 -3904.175} C_VEL
LIN {X 0,Y 538.007,Z 457.469,A -85,B 0,C 180,E1 -3907.171,E2 -3907.171} C_VEL
LIN {X 0,Y 538.025,Z 457.46,A -85,B 0,C 180,E1 -3909.798,E2 -3909.798} C_VEL
LIN {X 0,Y 538.023,Z 457.467,A -85,B 0,C 180,E1 -3912.787,E2 -3912.787} C_VEL
LIN {X 0,Y 538.022,Z 457.462,A -85,B 0,C 180,E1 -3915.928,E2 -3915.928} C_VEL
LIN {X 0,Y 538.035,Z 457.463,A -85,B 0,C 180,E1 -3918.227,E2 -3918.227} C_VEL
LIN {X 0,Y 538.015,Z 457.468,A -85,B 0,C 180,E1 -3921.17,E2 -3921.17} C_VEL
LIN {X 0,Y 538.063,Z 457.65,A -85,B 0,C 180,E1 -3923.289,E2 -3923.289} C_VEL
LIN {X 0,Y 539.22,Z 463.949,A -85,B 0,C 180,E1 -3924.321,E2 -3924.321} C_VEL
LIN {X 0,Y 539.113,Z 476.986,A -85,B 0,C 180,E1 -3926.317,E2 -3926.317} C_VEL
LIN {X 0,Y 538.744,Z 495.927,A -85,B 0,C 180,E1 -3929.202,E2 -3929.202} C_VEL
LIN {X 0,Y 538.375,Z 514.543,A -85,B 0,C 180,E1 -3932.051,E2 -3932.051} C_VEL
LIN {X 0,Y 538.512,Z 517.127,A -85,B 0,C 180,E1 -3932.309,E2 -3932.309} C_VEL
LIN {X 0,Y 539.697,Z 525.56,A -85,B 0,C 180,E1 -3932.462,E2 -3932.462} C_VEL
LIN {X 0,Y 539.293,Z 623.678,A -85,B 0,C 180,E1 -3933.793,E2 -3933.793} C_VEL
LIN {X 0,Y 539.136,Z 636.651,A -85,B 0,C 180,E1 -3934.101,E2 -3934.101} C_VEL
LIN {X 0,Y 538.904,Z 649.041,A -85,B 0,C 180,E1 -3934.561,E2 -3934.561} C_VEL
LIN {X 0,Y 538.794,Z 658.482,A -85,B 0,C 180,E1 -3935.021,E2 -3935.021} C_VEL
LIN {X 0,Y 538.573,Z 668.448,A -85,B 0,C 180,E1 -3935.618,E2 -3935.618} C_VEL
LIN {X 0,Y 538.342,Z 679.463,A -85,B 0,C 180,E1 -3936.434,E2 -3936.434} C_VEL
LIN {X 0,Y 538.114,Z 689.128,A -85,B 0,C 180,E1 -3937.339,E2 -3937.339} C_VEL
LIN {X 0,Y 537.962,Z 696.302,A -85,B 0,C 180,E1 -3938.14,E2 -3938.14} C_VEL
LIN {X 0,Y 537.809,Z 703.822,A -85,B 0,C 180,E1 -3939.14,E2 -3939.14} C_VEL
LIN {X 0,Y 537.708,Z 710.581,A -85,B 0,C 180,E1 -3940.233,E2 -3940.233} C_VEL
LIN {X 0,Y 537.619,Z 715.934,A -85,B 0,C 180,E1 -3941.321,E2 -3941.321} C_VEL
LIN {X 0,Y 537.551,Z 720.483,A -85,B 0,C 180,E1 -3942.5,E2 -3942.5} C_VEL
LIN {X 0,Y 537.528,Z 722.9,A -85,B 0,C 180,E1 -3943.283,E2 -3943.283} C_VEL
LIN {X 0,Y 537.463,Z 724.841,A -85,B 0,C 180,E1 -3944.062,E2 -3944.062} C_VEL
LIN {X 0,Y 537.454,Z 726.979,A -85,B 0,C 180,E1 -3945.392,E2 -3945.392} C_VEL
LIN {X 0,Y 537.472,Z 727.794,A -85,B 0,C 180,E1 -3946.387,E2 -3946.387} C_VEL
LIN {X 0,Y 537.476,Z 727.983,A -85,B 0,C 180,E1 -3947.157,E2 -3947.157} C_VEL
LIN {X 0,Y 537.474,Z 727.713,A -85,B 0,C 180,E1 -3947.924,E2 -3947.924} C_VEL
LIN {X 0,Y 537.545,Z 726.983,A -85,B 0,C 180,E1 -3948.69,E2 -3948.69} C_VEL
LIN {X 0,Y 537.5,Z 724.411,A -85,B 0,C 180,E1 -3950.214,E2 -3950.214} C_VEL
LIN {X 0,Y 537.575,Z 721.269,A -85,B 0,C 180,E1 -3951.353,E2 -3951.353} C_VEL
LIN {X 0,Y 537.62,Z 717.099,A -85,B 0,C 180,E1 -3952.489,E2 -3952.489} C_VEL
LIN {X 0,Y 537.683,Z 711.718,A -85,B 0,C 180,E1 -3953.639,E2 -3953.639} C_VEL
LIN {X 0,Y 537.746,Z 703.904,A -85,B 0,C 180,E1 -3954.939,E2 -3954.939} C_VEL
LIN {X 0,Y 537.927,Z 696.883,A -85,B 0,C 180,E1 -3955.88,E2 -3955.88} C_VEL
LIN {X 0,Y 538.121,Z 688.492,A -85,B 0,C 180,E1 -3956.818,E2 -3956.818} C_VEL
LIN {X 0,Y 538.365,Z 678.21,A -85,B 0,C 180,E1 -3957.756,E2 -3957.756} C_VEL
LIN {X 0,Y 538.54,Z 667.96,A -85,B 0,C 180,E1 -3958.505,E2 -3958.505} C_VEL
LIN {X 0,Y 538.742,Z 658.574,A -85,B 0,C 180,E1 -3959.066,E2 -3959.066} C_VEL
LIN {X 0,Y 539.018,Z 646.809,A -85,B 0,C 180,E1 -3959.627,E2 -3959.627} C_VEL
LIN {X 0,Y 539.185,Z 634.448,A -85,B 0,C 180,E1 -3960.047,E2 -3960.047} C_VEL
LIN {X 0,Y 539.3,Z 623.317,A -85,B 0,C 180,E1 -3960.304,E2 -3960.304} C_VEL
LIN {X 0,Y 539.538,Z 523.805,A -85,B 0,C 180,E1 -3961.656,E2 -3961.656} C_VEL
LIN {X 0,Y 538.485,Z 516.847,A -85,B 0,C 180,E1 -3961.8,E2 -3961.8} C_VEL
LIN {X 0,Y 538.418,Z 514.481,A -85,B 0,C 180,E1 -3962.057,E2 -3962.057} C_VEL
LIN {X 0,Y 538.691,Z 497.497,A -85,B 0,C 180,E1 -3964.677,E2 -3964.677} C_VEL
LIN {X 0,Y 538.986,Z 481.313,A -85,B 0,C 180,E1 -3967.116,E2 -3967.116} C_VEL
LIN {X 0,Y 539.211,Z 466.38,A -85,B 0,C 180,E1 -3969.377,E2 -3969.377} C_VEL
LIN {X 0,Y 538.985,Z 462.543,A -85,B 0,C 180,E1 -3969.949,E2 -3969.949} C_VEL
LIN {X 0,Y 538.087,Z 457.561,A -85,B 0,C 180,E1 -3970.751,E2 -3970.751} C_VEL
LIN {X 0,Y 538.004,Z 457.47,A -85,B 0,C 180,E1 -3973.6,E2 -3973.6} C_VEL
LIN {X 0,Y 537.995,Z 457.468,A -85,B 0,C 180,E1 -3975.922,E2 -3975.922} C_VEL
LIN {X 0,Y 538.015,Z 457.465,A -85,B 0,C 180,E1 -3978.271,E2 -3978.271} C_VEL
LIN {X 0,Y 538.043,Z 457.464,A -85,B 0,C 180,E1 -3980.652,E2 -3980.652} C_VEL
LIN {X 0,Y 538.014,Z 457.464,A -85,B 0,C 180,E1 -3983.878,E2 -3983.878} C_VEL
LIN {X 0,Y 538.043,Z 457.462,A -85,B 0,C 180,E1 -3986.367,E2 -3986.367} C_VEL
LIN {X 0,Y 538.038,Z 457.468,A -85,B 0,C 180,E1 -3988.933,E2 -3988.933} C_VEL
LIN {X 0,Y 538.019,Z 457.463,A -85,B 0,C 180,E1 -3991.887,E2 -3991.887} C_VEL
LIN {X 0,Y 538.021,Z 457.469,A -85,B 0,C 180,E1 -3994.617,E2 -3994.617} C_VEL
LIN {X 0,Y 538.012,Z 457.466,A -85,B 0,C 180,E1 -3997.17,E2 -3997.17} C_VEL
LIN {X 0,Y 538.031,Z 457.462,A -85,B 0,C 180,E1 -3999.797,E2 -3999.797} C_VEL
LIN {X 0,Y 538.027,Z 457.467,A -85,B 0,C 180,E1 -4002.786,E2 -4002.786} C_VEL
LIN {X 0,Y 538.026,Z 457.465,A -85,B 0,C 180,E1 -4005.926,E2 -4005.926} C_VEL
LIN {X 0,Y 538.038,Z 457.468,A -85,B 0,C 180,E1 -4008.226,E2 -4008.226} C_VEL
LIN {X 0,Y 538.018,Z 457.458,A -85,B 0,C 180,E1 -4011.169,E2 -4011.169} C_VEL
LIN {X 0,Y 537.995,Z 457.473,A -85,B 0,C 180,E1 -4014.089,E2 -4014.089} C_VEL
LIN {X 0,Y 538.038,Z 457.464,A -85,B 0,C 180,E1 -4016.727,E2 -4016.727} C_VEL
LIN {X 0,Y 538.02,Z 457.467,A -85,B 0,C 180,E1 -4019.558,E2 -4019.558} C_VEL
LIN {X 0,Y 538.048,Z 457.682,A -85,B 0,C 180,E1 -4021.896,E2 -4021.896} C_VEL
LIN {X 0,Y 540.392,Z 468.905,A -85,B 0,C 180,E1 -4023.34,E2 -4023.34} C_VEL
LIN {X 0,Y 539.966,Z 490.942,A -85,B 0,C 180,E1 -4025.904,E2 -4025.904} C_VEL
LIN {X 0,Y 539.646,Z 513.002,A -85,B 0,C 180,E1 -4028.412,E2 -4028.412} C_VEL
LIN {X 0,Y 539.18,Z 541.24,A -85,B 0,C 180,E1 -4031.572,E2 -4031.572} C_VEL
LIN {X 0,Y 538.779,Z 567.377,A -85,B 0,C 180,E1 -4034.489,E2 -4034.489} C_VEL
LIN {X 0,Y 538.695,Z 573.871,A -85,B 0,C 180,E1 -4035.213,E2 -4035.213} C_VEL
LIN {X 0,Y 539.723,Z 582.15,A -85,B 0,C 180,E1 -4035.371,E2 -4035.371} C_VEL
LIN {X 0,Y 539.328,Z 683.89,A -85,B 0,C 180,E1 -4036.745,E2 -4036.745} C_VEL
LIN {X 0,Y 539.173,Z 696.418,A -85,B 0,C 180,E1 -4037.053,E2 -4037.053} C_VEL
LIN {X 0,Y 538.991,Z 709.341,A -85,B 0,C 180,E1 -4037.527,E2 -4037.527} C_VEL
LIN {X 0,Y 538.79,Z 720.768,A -85,B 0,C 180,E1 -4038.095,E2 -4038.095} C_VEL
LIN {X 0,Y 538.54,Z 731.887,A -85,B 0,C 180,E1 -4038.805,E2 -4038.805} C_VEL
LIN {X 0,Y 538.309,Z 742.523,A -85,B 0,C 180,E1 -4039.657,E2 -4039.657} C_VEL
LIN {X 0,Y 538.069,Z 752.102,A -85,B 0,C 180,E1 -4040.602,E2 -4040.602} C_VEL
LIN {X 0,Y 537.92,Z 759.951,A -85,B 0,C 180,E1 -4041.547,E2 -4041.547} C_VEL
LIN {X 0,Y 537.756,Z 767.615,A -85,B 0,C 180,E1 -4042.678,E2 -4042.678} C_VEL
LIN {X 0,Y 537.694,Z 774.674,A -85,B 0,C 180,E1 -4043.997,E2 -4043.997} C_VEL
LIN {X 0,Y 537.541,Z 779.368,A -85,B 0,C 180,E1 -4045.124,E2 -4045.124} C_VEL
LIN {X 0,Y 537.591,Z 782.955,A -85,B 0,C 180,E1 -4046.251,E2 -4046.251} C_VEL
LIN {X 0,Y 537.551,Z 784.804,A -85,B 0,C 180,E1 -4047.001,E2 -4047.001} C_VEL
LIN {X 0,Y 537.451,Z 787.182,A -85,B 0,C 180,E1 -4048.5,E2 -4048.5} C_VEL
LIN {X 0,Y 537.442,Z 788,A -85,B 0,C 180,E1 -4049.999,E2 -4049.999} C_VEL
LIN {X 0,Y 537.451,Z 787.186,A -85,B 0,C 180,E1 -4051.497,E2 -4051.497} C_VEL
LIN {X 0,Y 537.551,Z 784.813,A -85,B 0,C 180,E1 -4052.996,E2 -4052.996} C_VEL
LIN {X 0,Y 537.603,Z 781.899,A -85,B 0,C 180,E1 -4054.122,E2 -4054.122} C_VEL
LIN {X 0,Y 537.587,Z 777.953,A -85,B 0,C 180,E1 -4055.249,E2 -4055.249} C_VEL
LIN {X 0,Y 537.642,Z 773.136,A -85,B 0,C 180,E1 -4056.324,E2 -4056.324} C_VEL
LIN {X 0,Y 537.79,Z 766.475,A -85,B 0,C 180,E1 -4057.508,E2 -4057.508} C_VEL
LIN {X 0,Y 537.971,Z 758.488,A -85,B 0,C 180,E1 -4058.639,E2 -4058.639} C_VEL
LIN {X 0,Y 538.144,Z 750.346,A -85,B 0,C 180,E1 -4059.584,E2 -4059.584} C_VEL
LIN {X 0,Y 538.342,Z 740.413,A -85,B 0,C 180,E1 -4060.53,E2 -4060.53} C_VEL
LIN {X 0,Y 538.577,Z 730.611,A -85,B 0,C 180,E1 -4061.286,E2 -4061.286} C_VEL
LIN {X 0,Y 538.803,Z 719.721,A -85,B 0,C 180,E1 -4061.962,E2 -4061.962} C_VEL
LIN {X 0,Y 538.994,Z 707.135,A -85,B 0,C 180,E1 -4062.566,E2 -4062.566} C_VEL
LIN {X 0,Y 539.193,Z 694.139,A -85,B 0,C 180,E1 -4063.016,E2 -4063.016} C_VEL
LIN {X 0,Y 539.358,Z 681.191,A -85,B 0,C 180,E1 -4063.3,E2 -4063.3} C_VEL
LIN {X 0,Y 539.542,Z 580.33,A -85,B 0,C 180,E1 -4064.658,E2 -4064.658} C_VEL
LIN {X 0,Y 538.704,Z 573.948,A -85,B 0,C 180,E1 -4064.785,E2 -4064.785} C_VEL
LIN {X 0,Y 539.119,Z 545.277,A -85,B 0,C 180,E1 -4067.998,E2 -4067.998} C_VEL
LIN {X 0,Y 539.576,Z 518.703,A -85,B 0,C 180,E1 -4070.987,E2 -4070.987} C_VEL
LIN {X 0,Y 540.033,Z 491.396,A -85,B 0,C 180,E1 -4074.098,E2 -4074.098} C_VEL
LIN {X 0,Y 540.438,Z 469.593,A -85,B 0,C 180,E1 -4076.655,E2 -4076.655} C_VEL
LIN {X 0,Y 539.942,Z 466.021,A -85,B 0,C 180,E1 -4077.1,E2 -4077.1} C_VEL
LIN {X 0,Y 538.034,Z 457.64,A -85,B 0,C 180,E1 -4078.208,E2 -4078.208} C_VEL
LIN {X 0,Y 538.002,Z 457.47,A -85,B 0,C 180,E1 -4080.626,E2 -4080.626} C_VEL
LIN {X 0,Y 538.014,Z 457.465,A -85,B 0,C 180,E1 -4083.277,E2 -4083.277} C_VEL
LIN {X 0,Y 537.98,Z 457.475,A -85,B 0,C 180,E1 -4086.004,E2 -4086.004} C_VEL
LIN {X 0,Y 538.001,Z 457.465,A -85,B 0,C 180,E1 -4088.829,E2 -4088.829} C_VEL
LIN {X 0,Y 537.991,Z 457.469,A -85,B 0,C 180,E1 -4091.874,E2 -4091.874} C_VEL
LIN {X 0,Y 537.988,Z 457.466,A -85,B 0,C 180,E1 -4094.862,E2 -4094.862} C_VEL
LIN {X 0,Y 537.989,Z 457.465,A -85,B 0,C 180,E1 -4097.211,E2 -4097.211} C_VEL
LIN {X 0,Y 538,Z 457.473,A -85,B 0,C 180,E1 -4100.201,E2 -4100.201} C_VEL
LIN {X 0,Y 538.007,Z 457.463,A -85,B 0,C 180,E1 -4103.065,E2 -4103.065} C_VEL
LIN {X 0,Y 538.006,Z 457.466,A -85,B 0,C 180,E1 -4105.825,E2 -4105.825} C_VEL
LIN {X 0,Y 537.997,Z 457.471,A -85,B 0,C 180,E1 -4108.498,E2 -4108.498} C_VEL
LIN {X 0,Y 538.006,Z 457.463,A -85,B 0,C 180,E1 -4111.096,E2 -4111.096} C_VEL
LIN {X 0,Y 538.022,Z 457.461,A -85,B 0,C 180,E1 -4113.632,E2 -4113.632} C_VEL
LIN {X 0,Y 537.993,Z 457.47,A -85,B 0,C 180,E1 -4116.121,E2 -4116.121} C_VEL
LIN {X 0,Y 538.024,Z 457.46,A -85,B 0,C 180,E1 -4119.348,E2 -4119.348} C_VEL
LIN {X 0,Y 538.041,Z 457.467,A -85,B 0,C 180,E1 -4122.516,E2 -4122.516} C_VEL
LIN {X 0,Y 538.042,Z 457.459,A -85,B 0,C 180,E1 -4125.63,E2 -4125.63} C_VEL
LIN {X 0,Y 538.078,Z 457.46,A -85,B 0,C 180,E1 -4128.701,E2 -4128.701} C_VEL
LIN {X 0,Y 538.066,Z 457.456,A -85,B 0,C 180,E1 -4131.739,E2 -4131.739} C_VEL
LIN {X 0,Y 538.143,Z 457.452,A -85,B 0,C 180,E1 -4134.755,E2 -4134.755} C_VEL
